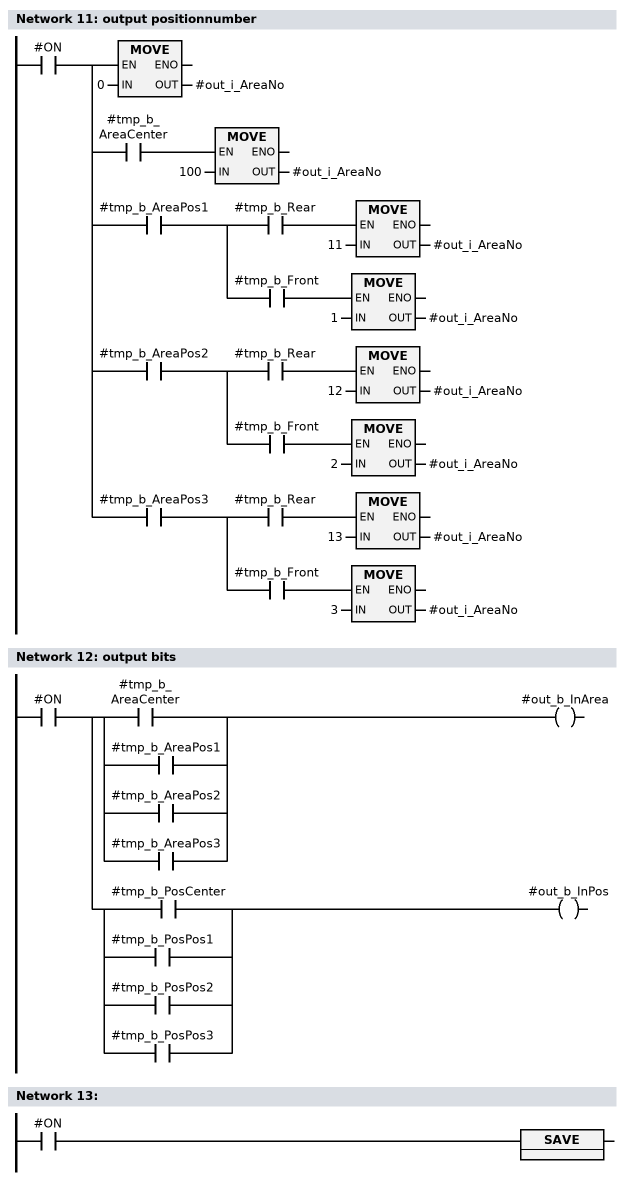
NETWORK
TITLE = output positionnumber
      A     #ON;
      =     L 10.0;
      A     L 10.0;
      JNB   _003;
      L     0;
      T     #out_i_AreaNo;
_003: NOP   0;
      A     L 10.0;
      A     #tmp_b_AreaCenter;
      JNB   _004;
      L     100;
      T     #out_i_AreaNo;
_004: NOP   0;
      A     L 10.0;
      A     #tmp_b_AreaPos1;
      =     L 10.1;
      A     L 10.1;
      A     #tmp_b_Rear;
      JNB   _005;
      L     11;
      T     #out_i_AreaNo;
_005: NOP   0;
      A     L 10.1;
      A     #tmp_b_Front;
      JNB   _006;
      L     1;
      T     #out_i_AreaNo;
_006: NOP   0;
      A     L 10.0;
      A     #tmp_b_AreaPos2;
      =     L 10.1;
      A     L 10.1;
      A     #tmp_b_Rear;
      JNB   _007;
      L     12;
      T     #out_i_AreaNo;
_007: NOP   0;
      A     L 10.1;
      A     #tmp_b_Front;
      JNB   _008;
      L     2;
      T     #out_i_AreaNo;
_008: NOP   0;
      A     L 10.0;
      A     #tmp_b_AreaPos3;
      =     L 10.1;
      A     L 10.1;
      A     #tmp_b_Rear;
      JNB   _009;
      L     13;
      T     #out_i_AreaNo;
_009: NOP   0;
      A     L 10.1;
      A     #tmp_b_Front;
      JNB   _00a;
      L     3;
      T     #out_i_AreaNo;
_00a: NOP   0;
NETWORK
TITLE = output bits
      A     #ON;
      =     L 10.0;
      A     L 10.0;
      A(;
      O     #tmp_b_AreaCenter;
      O     #tmp_b_AreaPos1;
      O     #tmp_b_AreaPos2;
      O     #tmp_b_AreaPos3;
      );
      =     #out_b_InArea;
      A     L 10.0;
      A(;
      O     #tmp_b_PosCenter;
      O     #tmp_b_PosPos1;
      O     #tmp_b_PosPos2;
      O     #tmp_b_PosPos3;
      );
      =     #out_b_InPos;
NETWORK
TITLE =
      A     #ON;
      SAVE;
END_FUNCTION

FUNCTION "Scan_TEL_Man" : VOID	// FC 28
TITLE = scan positions TELescopes manual mode
VERSION : 1.0
VAR_INPUT
  in_i_DBNo : INT ;
  in_i_NoOfDataSets : INT ;
  in_i_DatSetLenght : INT ;
  in_i_DataStartByte : INT ;
  in_di_ActAxisPos : DINT ;
  in_di_PosValMin : DINT ;
  in_di_PosValMax : DINT ;
END_VAR
VAR_OUTPUT
  out_di_PrevPos : DINT ;
  out_di_ActPos : DINT ;
  out_di_NextPos : DINT ;
  out_di_MinPos : DINT ;
  out_di_MaxPos : DINT ;
END_VAR
VAR_TEMP
  tmp_di_1 : DINT ;
  tmp_di_Pointer : DINT ;
  tmp_di_ChkPosVal : DINT ;
  tmp_di_PosData : DINT ;
  tmp_di_PosDataPlus : DINT ;
  tmp_di_PosDataMinus : DINT ;
  tmp_di_PosDataLow : DINT ;
  tmp_di_PosDataHigh : DINT ;
  tmp_di_PrevPos : DINT ;
  tmp_di_NextPos : DINT ;
  tmp_di_MinPos : DINT ;
  tmp_di_MaxPos : DINT ;
  tmp_di_TEL_in : DINT ;
  tmp_di_TEL_mid : DINT ;
  tmp_di_TEL_out : DINT ;
  tmp_i_NoOfDataSets : INT ;
  tmp_i_Counter : INT ;
  tmp_i_DBNo : INT ;
  ON : BOOL ;
  OFF : BOOL ;
END_VAR
BEGIN
NETWORK
TITLE = on/off
      SET;
      =     #ON;
      CLR;
      =     #OFF;
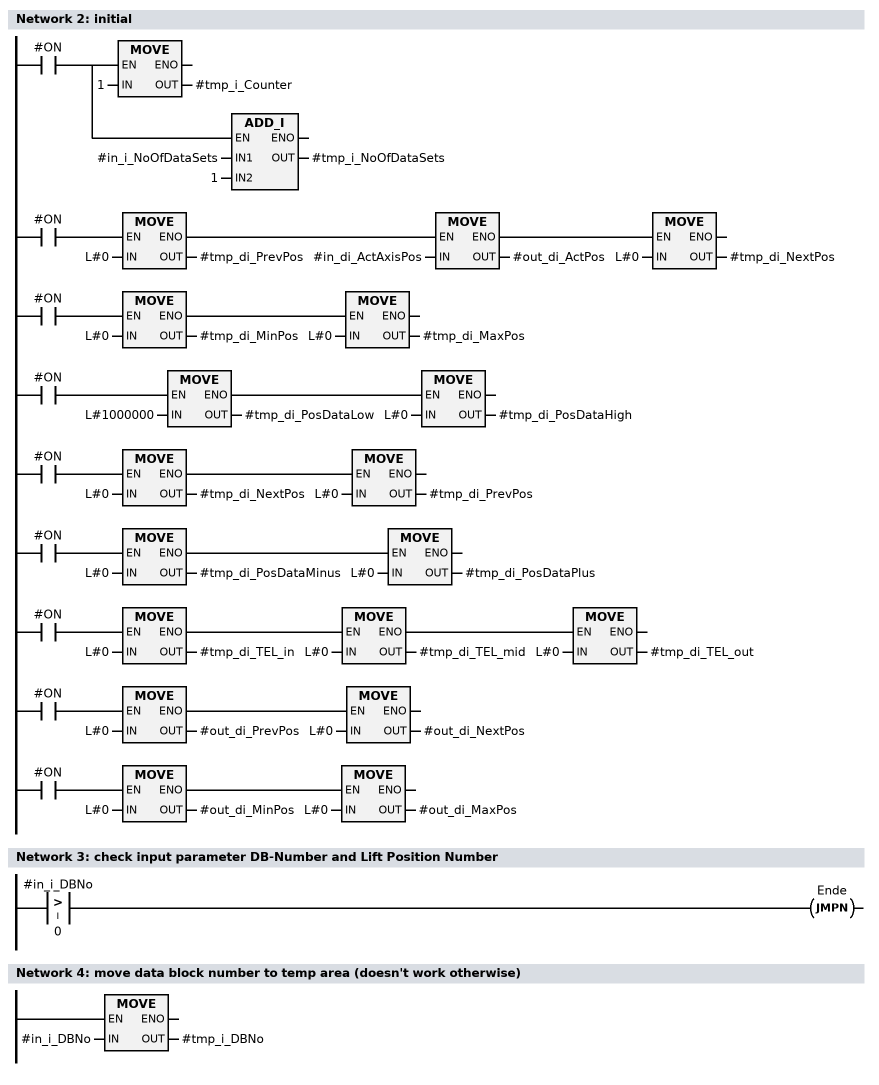
NETWORK
TITLE = initial
//set loopcounter to 0
//reset outputs
      A     #ON;
      =     L 67.0;
      A     L 67.0;
      JNB   _001;
      L     1;
      T     #tmp_i_Counter;
_001: NOP   0;
      A(;
      A(;
      A     L 67.0;
      JNB   _002;
      L     L#0;
      T     #tmp_di_PrevPos;
      SET;
      SAVE;
      CLR;
_002: A     BR;
      );
      JNB   _003;
      L     #in_di_ActAxisPos;
      T     #out_di_ActPos;
      SET;
      SAVE;
      CLR;
_003: A     BR;
      );
      JNB   _004;
      L     L#0;
      T     #tmp_di_NextPos;
_004: NOP   0;
      A(;
      A     L 67.0;
      JNB   _005;
      L     L#0;
      T     #tmp_di_MinPos;
      SET;
      SAVE;
      CLR;
_005: A     BR;
      );
      JNB   _006;
      L     L#0;
      T     #tmp_di_MaxPos;
_006: NOP   0;
      A(;
      A     L 67.0;
      JNB   _007;
      L     L#1000000;
      T     #tmp_di_PosDataLow;
      SET;
      SAVE;
      CLR;
_007: A     BR;
      );
      JNB   _008;
      L     L#0;
      T     #tmp_di_PosDataHigh;
_008: NOP   0;
      A(;
      A     L 67.0;
      JNB   _009;
      L     L#0;
      T     #tmp_di_NextPos;
      SET;
      SAVE;
      CLR;
_009: A     BR;
      );
      JNB   _00a;
      L     L#0;
      T     #tmp_di_PrevPos;
_00a: NOP   0;
      A(;
      A     L 67.0;
      JNB   _00b;
      L     L#0;
      T     #tmp_di_PosDataMinus;
      SET;
      SAVE;
      CLR;
_00b: A     BR;
      );
      JNB   _00c;
      L     L#0;
      T     #tmp_di_PosDataPlus;
_00c: NOP   0;
      A(;
      A(;
      A     L 67.0;
      JNB   _00d;
      L     L#0;
      T     #tmp_di_TEL_in;
      SET;
      SAVE;
      CLR;
_00d: A     BR;
      );
      JNB   _00e;
      L     L#0;
      T     #tmp_di_TEL_mid;
      SET;
      SAVE;
      CLR;
_00e: A     BR;
      );
      JNB   _00f;
      L     L#0;
      T     #tmp_di_TEL_out;
_00f: NOP   0;
      A     L 67.0;
      JNB   _010;
      L     #in_i_NoOfDataSets;
      L     1;
      +I;
      T     #tmp_i_NoOfDataSets;
_010: NOP   0;
      A(;
      A     L 67.0;
      JNB   _011;
      L     L#0;
      T     #out_di_PrevPos;
      SET;
      SAVE;
      CLR;
_011: A     BR;
      );
      JNB   _012;
      L     L#0;
      T     #out_di_NextPos;
_012: NOP   0;
      A(;
      A     L 67.0;
      JNB   _013;
      L     L#0;
      T     #out_di_MinPos;
      SET;
      SAVE;
      CLR;
_013: A     BR;
      );
      JNB   _014;
      L     L#0;
      T     #out_di_MaxPos;
_014: NOP   0;
NETWORK
TITLE = check input parameter DB-Number and Lift Position Number
//DB-Number > 0 and Lift in valid position
//or
//Lift position is intern hook
      L     #in_i_DBNo;
      L     0;
      >I;
      JCN   Ende;
NETWORK
TITLE = move data block number to temp area (doesn't work otherwise)
//doesn't work otherwise
      L     #in_i_DBNo;
      T     #tmp_i_DBNo;
      NOP   0;
NETWORK
TITLE = open DB
      OPN   DB [#tmp_i_DBNo];
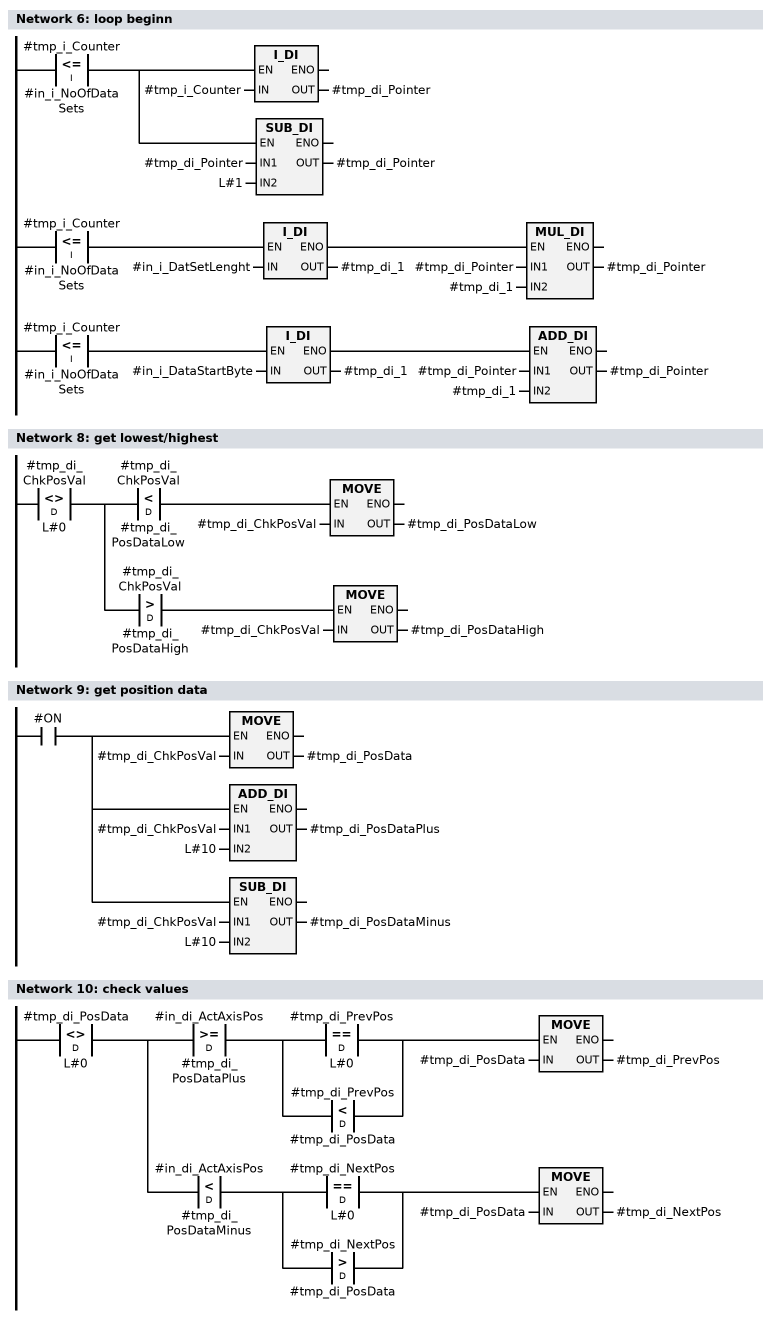
NETWORK
TITLE = loop beginn
//calculate pointer to positionvalue
scbr: L     #tmp_i_Counter;
      L     #in_i_NoOfDataSets;
      <=I;
      =     L 67.0;
      A     L 67.0;
      JNB   _015;
      L     #tmp_i_Counter;
      ITD;
      T     #tmp_di_Pointer;
_015: NOP   0;
      A     L 67.0;
      JNB   _016;
      L     #tmp_di_Pointer;
      L     L#1;
      -D;
      T     #tmp_di_Pointer;
_016: NOP   0;
      A(;
      A     L 67.0;
      JNB   _017;
      L     #in_i_DatSetLenght;
      ITD;
      T     #tmp_di_1;
      SET;
      SAVE;
      CLR;
_017: A     BR;
      );
      JNB   _018;
      L     #tmp_di_Pointer;
      L     #tmp_di_1;
      *D;
      T     #tmp_di_Pointer;
_018: NOP   0;
      A(;
      A     L 67.0;
      JNB   _019;
      L     #in_i_DataStartByte;
      ITD;
      T     #tmp_di_1;
      SET;
      SAVE;
      CLR;
_019: A     BR;
      );
      JNB   _01a;
      L     #tmp_di_Pointer;
      L     #tmp_di_1;
      +D;
      T     #tmp_di_Pointer;
_01a: NOP   0;
NETWORK
TITLE = get positionvalue
      L     #tmp_di_Pointer;	// load pointer
      SLD   3;	// shift left 3 bits to achieve pointer format
      LAR1;	// load adressregister 1 with pointer
      L     DBD [AR1,P#0.0];	// load position from DataBlock
      T     #tmp_di_ChkPosVal;
NETWORK
TITLE = get lowest/highest
      L     #tmp_di_ChkPosVal;
      L     L#0;
      <>D;
      =     L 67.0;
      A     L 67.0;
      A(;
      L     #tmp_di_ChkPosVal;
      L     #tmp_di_PosDataLow;
      <D;
      );
      JNB   _01b;
      L     #tmp_di_ChkPosVal;
      T     #tmp_di_PosDataLow;
_01b: NOP   0;
      A     L 67.0;
      A(;
      L     #tmp_di_ChkPosVal;
      L     #tmp_di_PosDataHigh;
      >D;
      );
      JNB   _01c;
      L     #tmp_di_ChkPosVal;
      T     #tmp_di_PosDataHigh;
_01c: NOP   0;
NETWORK
TITLE = get position data
      A     #ON;
      =     L 67.0;
      A     L 67.0;
      JNB   _01d;
      L     #tmp_di_ChkPosVal;
      T     #tmp_di_PosData;
_01d: NOP   0;
      A     L 67.0;
      JNB   _01e;
      L     #tmp_di_ChkPosVal;
      L     L#10;
      +D;
      T     #tmp_di_PosDataPlus;
_01e: NOP   0;
      A     L 67.0;
      JNB   _01f;
      L     #tmp_di_ChkPosVal;
      L     L#10;
      -D;
      T     #tmp_di_PosDataMinus;
_01f: NOP   0;
NETWORK
TITLE = check values
      L     #tmp_di_PosData;
      L     L#0;
      <>D;
      =     L 67.0;
      A     L 67.0;
      A(;
      L     #in_di_ActAxisPos;
      L     #tmp_di_PosDataPlus;
      >=D;
      );
      A(;
      O(;
      L     #tmp_di_PrevPos;
      L     L#0;
      ==D;
      );
      O(;
      L     #tmp_di_PrevPos;
      L     #tmp_di_PosData;
      <D;
      );
      );
      JNB   _020;
      L     #tmp_di_PosData;
      T     #tmp_di_PrevPos;
_020: NOP   0;
      A     L 67.0;
      A(;
      L     #in_di_ActAxisPos;
      L     #tmp_di_PosDataMinus;
      <D;
      );
      A(;
      O(;
      L     #tmp_di_NextPos;
      L     L#0;
      ==D;
      );
      O(;
      L     #tmp_di_NextPos;
      L     #tmp_di_PosData;
      >D;
      );
      );
      JNB   _021;
      L     #tmp_di_PosData;
      T     #tmp_di_NextPos;
_021: NOP   0;
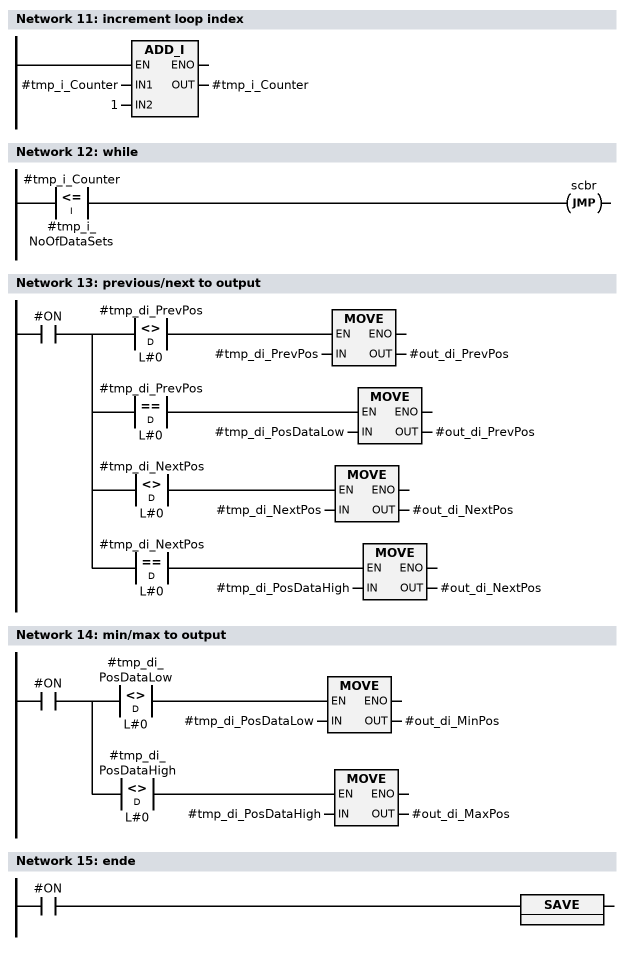
NETWORK
TITLE = increment loop index
      L     #tmp_i_Counter;
      L     1;
      +I;
      T     #tmp_i_Counter;
      NOP   0;
NETWORK
TITLE = while 
      L     #tmp_i_Counter;
      L     #tmp_i_NoOfDataSets;
      <=I;
      JC    scbr;
NETWORK
TITLE = previous/next to output
Ende: A     #ON;
      =     L 67.0;
      A     L 67.0;
      A(;
      L     #tmp_di_PrevPos;
      L     L#0;
      <>D;
      );
      JNB   _022;
      L     #tmp_di_PrevPos;
      T     #out_di_PrevPos;
_022: NOP   0;
      A     L 67.0;
      A(;
      L     #tmp_di_PrevPos;
      L     L#0;
      ==D;
      );
      JNB   _023;
      L     #tmp_di_PosDataLow;
      T     #out_di_PrevPos;
_023: NOP   0;
      A     L 67.0;
      A(;
      L     #tmp_di_NextPos;
      L     L#0;
      <>D;
      );
      JNB   _024;
      L     #tmp_di_NextPos;
      T     #out_di_NextPos;
_024: NOP   0;
      A     L 67.0;
      A(;
      L     #tmp_di_NextPos;
      L     L#0;
      ==D;
      );
      JNB   _025;
      L     #tmp_di_PosDataHigh;
      T     #out_di_NextPos;
_025: NOP   0;
NETWORK
TITLE = min/max to output
      A     #ON;
      =     L 67.0;
      A     L 67.0;
      A(;
      L     #tmp_di_PosDataLow;
      L     L#0;
      <>D;
      );
      JNB   _026;
      L     #tmp_di_PosDataLow;
      T     #out_di_MinPos;
_026: NOP   0;
      A     L 67.0;
      A(;
      L     #tmp_di_PosDataHigh;
      L     L#0;
      <>D;
      );
      JNB   _027;
      L     #tmp_di_PosDataHigh;
      T     #out_di_MaxPos;
_027: NOP   0;
NETWORK
TITLE = ende
      A     #ON;
      SAVE;
END_FUNCTION

FUNCTION "SCALE_WAGO_AI" : WORD	// FC 29
TITLE = SCALING VALUES
//Speziell für WAGO 250-466 4.20mA SE standard 
//Meßwertauflösung 12 bit (4095)
//
AUTHOR : SEA
FAMILY : CONVERT
NAME : SCALE
VERSION : 2.1
VAR_INPUT
  IN : INT ;	// input value to be scaled
  HI_LIM : REAL ;	// upper limit in engineering units
  LO_LIM : REAL ;	// lower limit in engineering units
  BIPOLAR : BOOL ;	// 1=bipolar; 0=unipolar
END_VAR
VAR_OUTPUT
  RET_VAL : WORD ;
  OUT : REAL ;	// result of the scale conversion
END_VAR
VAR_TEMP
  IN_REAL : REAL ;	// input value as a REAL number
  K1 : REAL ;	// low limit for input value
  K2 : REAL ;	// high limit for input value
  SPAN : REAL ;	// HI_LIM - LO_LIM
  TEMP1 : REAL ;	// temporary result
END_VAR
BEGIN
NETWORK
TITLE =
//
// set K1 and K2 constants based upon BIPOLAR
//
// (network holds code this reader does not know; not shown)
// convert input (IN) to real
// determine SPAN = HI_LIM - LO_LIM
// If the input value is outside the K1 and K2 range, the output
// is clamped to the nearer of either the LO_LIM or the HI_LIM 
// and an error is logged. If the input value is exactly at a limit the
// output will be set to the computed limit with no error returned.
//     changed 2/14/00 by ERI per RQ210693
// scale the input
// set BR bit : no error-set BR bit to 1; with error-set BR bit to 0.
END_FUNCTION

FUNCTION "Inputs" : VOID	// FC 30
TITLE = Inputs
VERSION : 0.1
VAR_TEMP
  tmp_Retval : INT ;
  tmp_d : INT ;
  tmp_u : DINT ;
  value : INT ;
  d_value : DINT ;
  ON : BOOL ;
  OFF : BOOL ;
  tmp_in : DINT ;
END_VAR
BEGIN
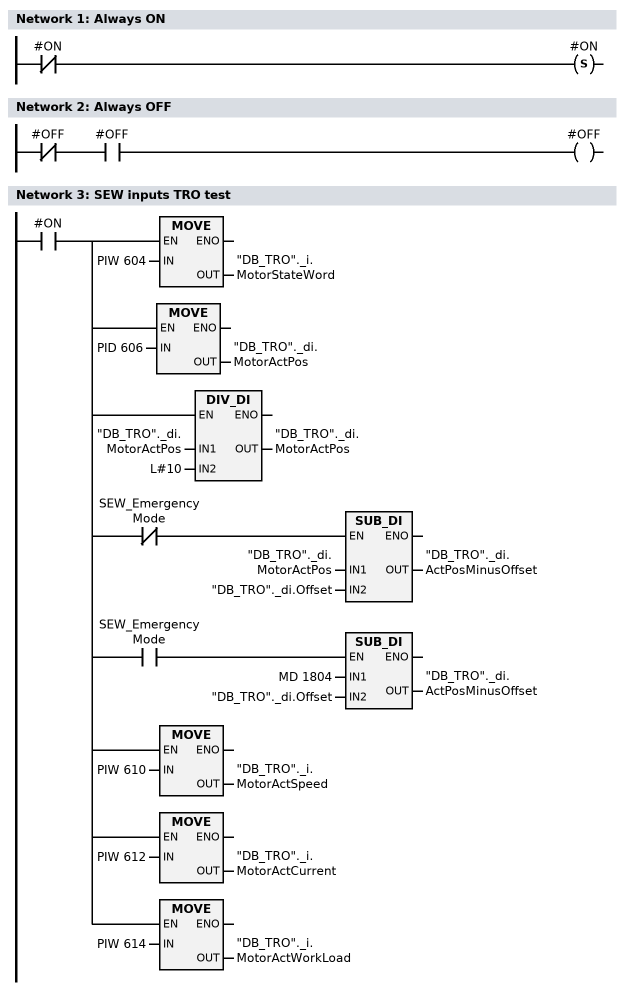
NETWORK
TITLE = Always ON
      AN    #ON;
      S     #ON;
NETWORK
TITLE = Always OFF
      AN    #OFF;
      A     #OFF;
      =     #OFF;
NETWORK
TITLE = SEW inputs TRO test
      A     #ON;
      =     L 20.0;
      A     L 20.0;
      JNB   _001;
      L     PIW 604;
      T     "DB_TRO"._i.MotorStateWord;
_001: NOP   0;
      A     L 20.0;
      JNB   _002;
      L     PID 606;
      T     "DB_TRO"._di.MotorActPos;
_002: NOP   0;
      A     L 20.0;
      JNB   _003;
      L     "DB_TRO"._di.MotorActPos;
      L     L#10;
      /D;
      T     "DB_TRO"._di.MotorActPos;
_003: NOP   0;
      A     L 20.0;
      AN    "SEW_EmergencyMode";
      JNB   _004;
      L     "DB_TRO"._di.MotorActPos;
      L     "DB_TRO"._di.Offset;
      -D;
      T     "DB_TRO"._di.ActPosMinusOffset;
_004: NOP   0;
      A     L 20.0;
      A     "SEW_EmergencyMode";
      JNB   _005;
      L     MD 1804;
      L     "DB_TRO"._di.Offset;
      -D;
      T     "DB_TRO"._di.ActPosMinusOffset;
_005: NOP   0;
      A     L 20.0;
      JNB   _006;
      L     PIW 610;
      T     "DB_TRO"._i.MotorActSpeed;
_006: NOP   0;
      A     L 20.0;
      JNB   _007;
      L     PIW 612;
      T     "DB_TRO"._i.MotorActCurrent;
_007: NOP   0;
      A     L 20.0;
      JNB   _008;
      L     PIW 614;
      T     "DB_TRO"._i.MotorActWorkLoad;
_008: NOP   0;
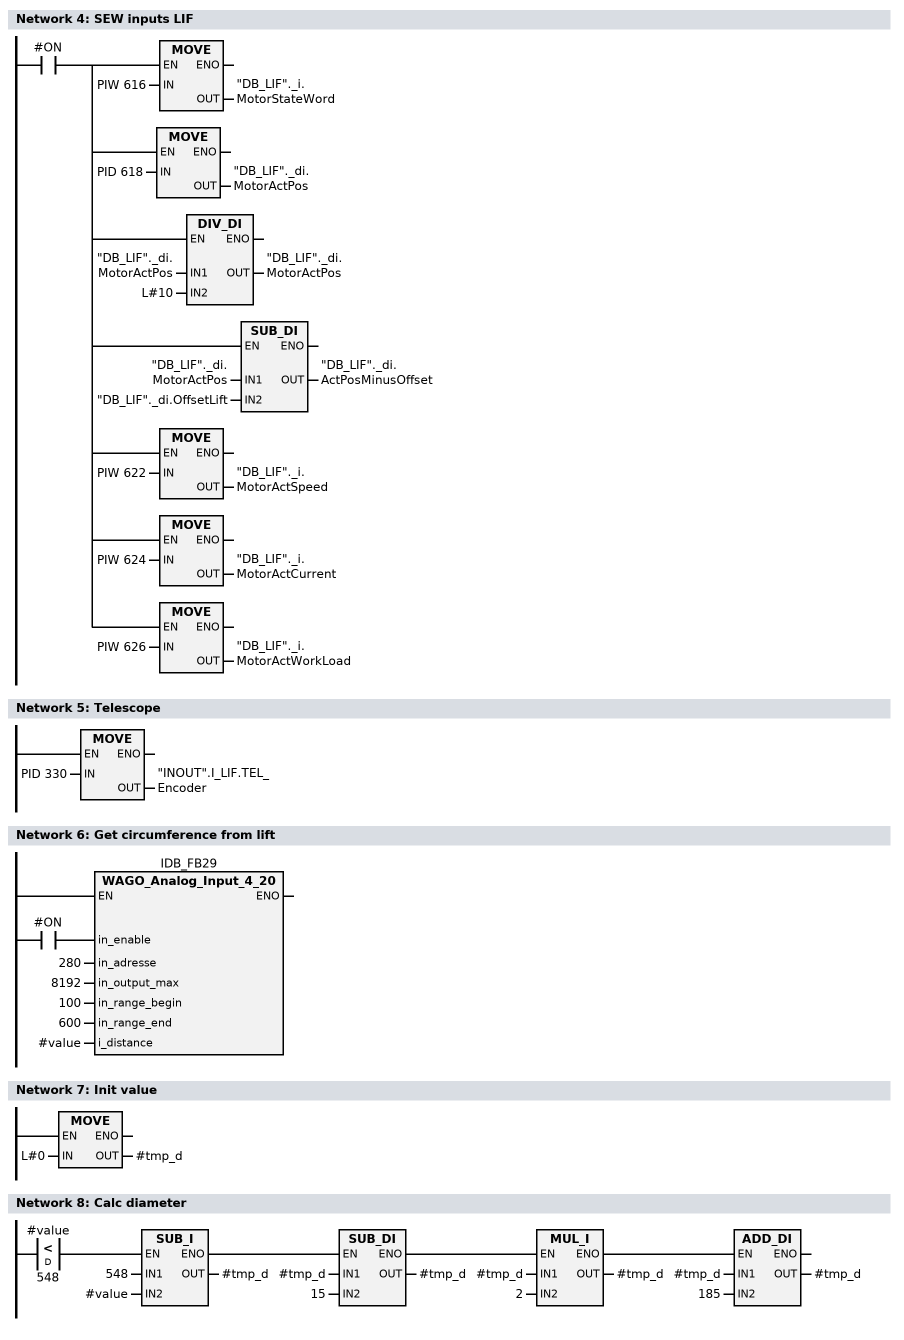
NETWORK
TITLE = SEW inputs LIF
      A     #ON;
      =     L 20.0;
      A     L 20.0;
      JNB   _009;
      L     PIW 616;
      T     "DB_LIF"._i.MotorStateWord;
_009: NOP   0;
      A     L 20.0;
      JNB   _00a;
      L     PID 618;
      T     "DB_LIF"._di.MotorActPos;
_00a: NOP   0;
      A     L 20.0;
      JNB   _00b;
      L     "DB_LIF"._di.MotorActPos;
      L     L#10;
      /D;
      T     "DB_LIF"._di.MotorActPos;
_00b: NOP   0;
      A     L 20.0;
      JNB   _00c;
      L     "DB_LIF"._di.MotorActPos;
      L     "DB_LIF"._di.OffsetLift;
      -D;
      T     "DB_LIF"._di.ActPosMinusOffset;
_00c: NOP   0;
      A     L 20.0;
      JNB   _00d;
      L     PIW 622;
      T     "DB_LIF"._i.MotorActSpeed;
_00d: NOP   0;
      A     L 20.0;
      JNB   _00e;
      L     PIW 624;
      T     "DB_LIF"._i.MotorActCurrent;
_00e: NOP   0;
      A     L 20.0;
      JNB   _00f;
      L     PIW 626;
      T     "DB_LIF"._i.MotorActWorkLoad;
_00f: NOP   0;
NETWORK
TITLE = Telescope
//we use a offset 10000
//
//bc17.02.2019: nachrüstung Encoder
//
      L     PID 330;
      T     "INOUT".I_LIF.TEL_Encoder;
      NOP   0;
NETWORK
TITLE = Get circumference from lift
//100mm = A1 Setpoint
//600mm = A2 Setpoint
//with pipe = 548
//US setting BEAM = 2
      A     #ON;
      =     L 20.0;
      BLD   103;
      CALL  "WAGO_Analog_Input_4_20" , "IDB_FB29" (
           in_enable                := L 20.0,
           in_adresse               := 280,
           in_output_max            := 8192,
           in_range_begin           := 100,
           in_range_end             := 600,
           i_distance               := #value);
      NOP   0;
NETWORK
TITLE = Init value
      L     L#0;
      T     #tmp_d;
      NOP   0;
NETWORK
TITLE = Calc diameter
//calc (548 - value - core thickness) * 2 + core diameter
      A(;
      A(;
      A(;
      A(;
      L     #value;
      L     548;
      <D;
      );
      JNB   _010;
      L     548;
      L     #value;
      -I;
      T     #tmp_d;
      AN    OV;
      SAVE;
      CLR;
_010: A     BR;
      );
      JNB   _011;
      L     #tmp_d;
      L     15;
      -D;
      T     #tmp_d;
      AN    OV;
      SAVE;
      CLR;
_011: A     BR;
      );
      JNB   _012;
      L     #tmp_d;
      L     2;
      *I;
      T     #tmp_d;
      AN    OV;
      SAVE;
      CLR;
_012: A     BR;
      );
      JNB   _013;
      L     #tmp_d;
      L     185;
      +D;
      T     #tmp_d;
_013: NOP   0;
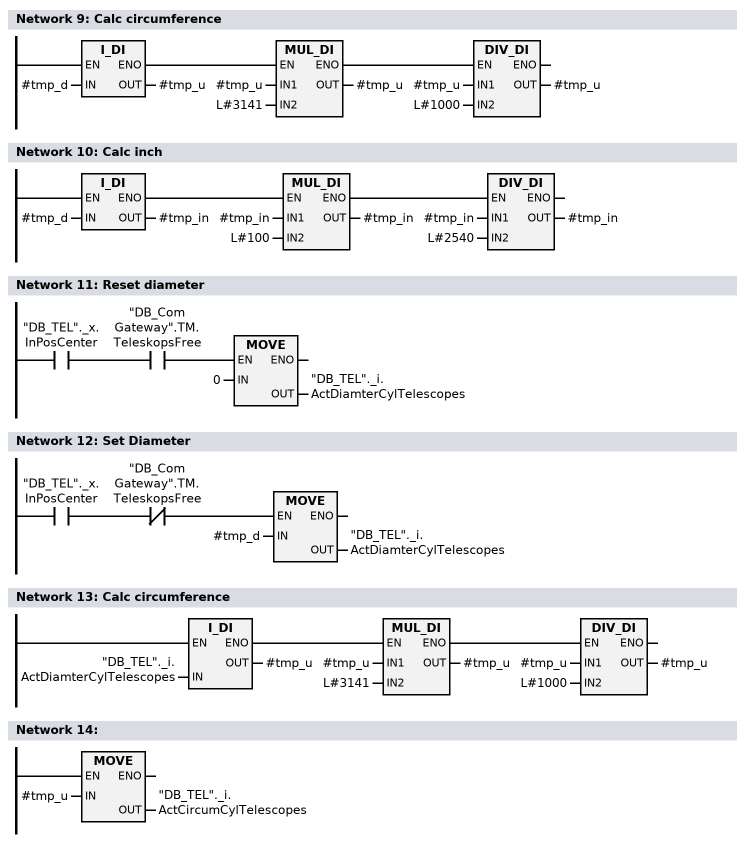
NETWORK
TITLE = Calc circumference
      A(;
      A(;
      L     #tmp_d;
      ITD;
      T     #tmp_u;
      SET;
      SAVE;
      CLR;
      A     BR;
      );
      JNB   _014;
      L     #tmp_u;
      L     L#3141;
      *D;
      T     #tmp_u;
      AN    OV;
      SAVE;
      CLR;
_014: A     BR;
      );
      JNB   _015;
      L     #tmp_u;
      L     L#1000;
      /D;
      T     #tmp_u;
_015: NOP   0;
NETWORK
TITLE = Calc inch
//25.4 mm = 1 inch 
//
//40 inch = 1016
//34 inch = 863
//14 inch = 355 330
      A(;
      A(;
      L     #tmp_d;
      ITD;
      T     #tmp_in;
      SET;
      SAVE;
      CLR;
      A     BR;
      );
      JNB   _016;
      L     #tmp_in;
      L     L#100;
      *D;
      T     #tmp_in;
      AN    OV;
      SAVE;
      CLR;
_016: A     BR;
      );
      JNB   _017;
      L     #tmp_in;
      L     L#2540;
      /D;
      T     #tmp_in;
_017: NOP   0;
NETWORK
TITLE = Reset diameter
      A     "DB_TEL"._x.InPosCenter;
      A     "DB_ComGateway".TM.TeleskopsFree;
      JNB   _018;
      L     0;
      T     "DB_TEL"._i.ActDiamterCylTelescopes;
_018: NOP   0;
NETWORK
TITLE = Set Diameter
      A     "DB_TEL"._x.InPosCenter;
      AN    "DB_ComGateway".TM.TeleskopsFree;
      JNB   _019;
      L     #tmp_d;
      T     "DB_TEL"._i.ActDiamterCylTelescopes;
_019: NOP   0;
NETWORK
TITLE = Calc circumference
      A(;
      A(;
      L     "DB_TEL"._i.ActDiamterCylTelescopes;
      ITD;
      T     #tmp_u;
      SET;
      SAVE;
      CLR;
      A     BR;
      );
      JNB   _01a;
      L     #tmp_u;
      L     L#3141;
      *D;
      T     #tmp_u;
      AN    OV;
      SAVE;
      CLR;
_01a: A     BR;
      );
      JNB   _01b;
      L     #tmp_u;
      L     L#1000;
      /D;
      T     #tmp_u;
_01b: NOP   0;
NETWORK
TITLE =
      L     #tmp_u;
      T     "DB_TEL"._i.ActCircumCylTelescopes;
      NOP   0;
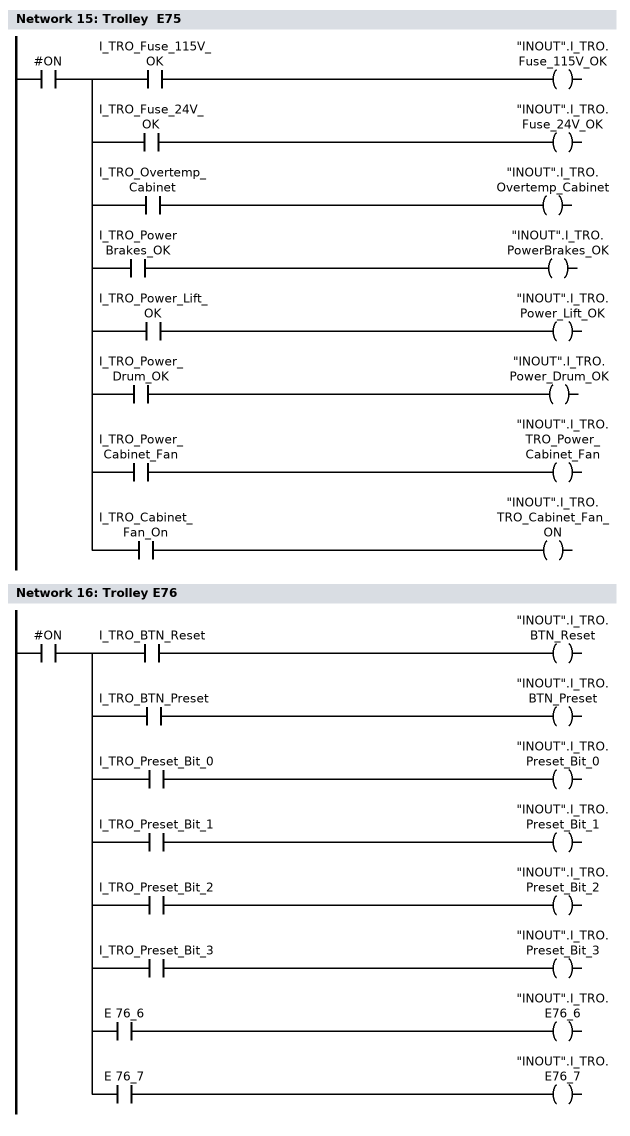
NETWORK
TITLE = Trolley  E75
      A     #ON;
      =     L 20.0;
      A     L 20.0;
      A     "I_TRO_Fuse_115V_OK";
      =     "INOUT".I_TRO.Fuse_115V_OK;
      A     L 20.0;
      A     "I_TRO_Fuse_24V_OK";
      =     "INOUT".I_TRO.Fuse_24V_OK;
      A     L 20.0;
      A     "I_TRO_Overtemp_Cabinet";
      =     "INOUT".I_TRO.Overtemp_Cabinet;
      A     L 20.0;
      A     "I_TRO_Power Brakes_OK";
      =     "INOUT".I_TRO.PowerBrakes_OK;
      A     L 20.0;
      A     "I_TRO_Power_Lift_OK";
      =     "INOUT".I_TRO.Power_Lift_OK;
      A     L 20.0;
      A     "I_TRO_Power_Drum_OK";
      =     "INOUT".I_TRO.Power_Drum_OK;
      A     L 20.0;
      A     "I_TRO_Power_Cabinet_Fan";
      =     "INOUT".I_TRO.TRO_Power_Cabinet_Fan;
      A     L 20.0;
      A     "I_TRO_Cabinet_Fan_On";
      =     "INOUT".I_TRO.TRO_Cabinet_Fan_ON;
NETWORK
TITLE = Trolley E76 
      A     #ON;
      =     L 20.0;
      A     L 20.0;
      A     "I_TRO_BTN_Reset";
      =     "INOUT".I_TRO.BTN_Reset;
      A     L 20.0;
      A     "I_TRO_BTN_Preset";
      =     "INOUT".I_TRO.BTN_Preset;
      A     L 20.0;
      A     "I_TRO_Preset_Bit_0";
      =     "INOUT".I_TRO.Preset_Bit_0;
      A     L 20.0;
      A     "I_TRO_Preset_Bit_1";
      =     "INOUT".I_TRO.Preset_Bit_1;
      A     L 20.0;
      A     "I_TRO_Preset_Bit_2";
      =     "INOUT".I_TRO.Preset_Bit_2;
      A     L 20.0;
      A     "I_TRO_Preset_Bit_3";
      =     "INOUT".I_TRO.Preset_Bit_3;
      A     L 20.0;
      A     "E 76_6";
      =     "INOUT".I_TRO.E76_6;
      A     L 20.0;
      A     "E 76_7";
      =     "INOUT".I_TRO.E76_7;
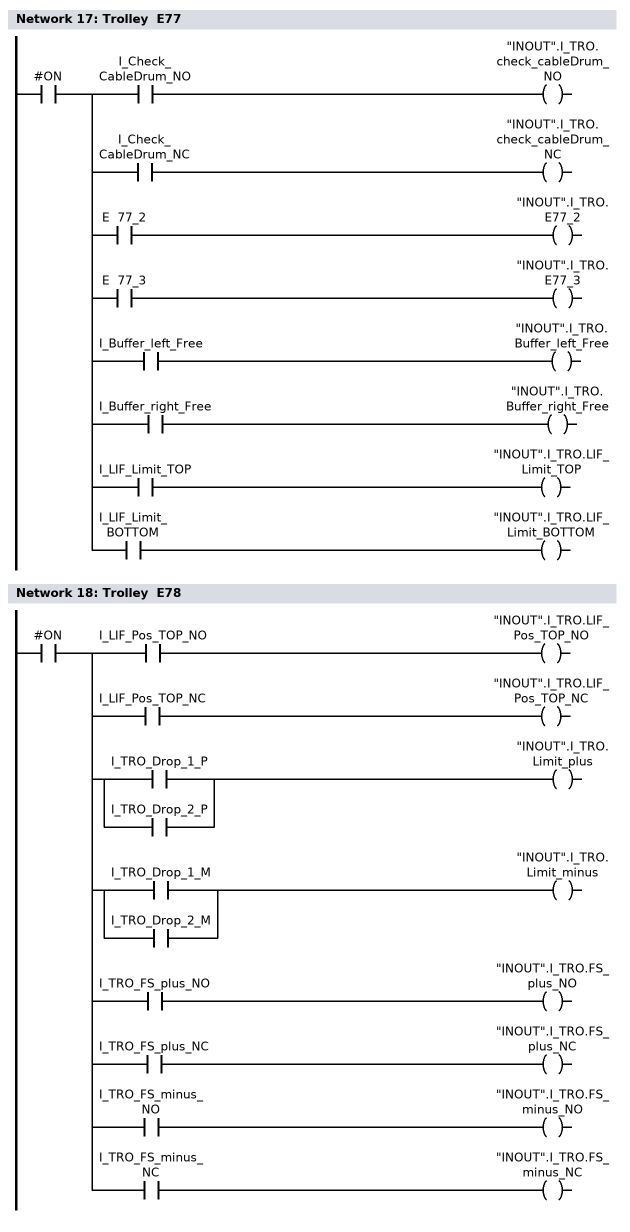
NETWORK
TITLE = Trolley  E77
      A     #ON;
      =     L 20.0;
      A     L 20.0;
      A     "I_Check_CableDrum_NO";
      =     "INOUT".I_TRO.check_cableDrum_NO;
      A     L 20.0;
      A     "I_Check_CableDrum_NC";
      =     "INOUT".I_TRO.check_cableDrum_NC;
      A     L 20.0;
      A     "E  77_2";
      =     "INOUT".I_TRO.E77_2;
      A     L 20.0;
      A     "E  77_3";
      =     "INOUT".I_TRO.E77_3;
      A     L 20.0;
      A     "I_Buffer_left_Free";
      =     "INOUT".I_TRO.Buffer_left_Free;
      A     L 20.0;
      A     "I_Buffer_right_Free";
      =     "INOUT".I_TRO.Buffer_right_Free;
      A     L 20.0;
      A     "I_LIF_Limit_TOP";
      =     "INOUT".I_TRO.LIF_Limit_TOP;
      A     L 20.0;
      A     "I_LIF_Limit_BOTTOM";
      =     "INOUT".I_TRO.LIF_Limit_BOTTOM;
NETWORK
TITLE = Trolley  E78
      A     #ON;
      =     L 20.0;
      A     L 20.0;
      A     "I_LIF_Pos_TOP_NO";
      =     "INOUT".I_TRO.LIF_Pos_TOP_NO;
      A     L 20.0;
      A     "I_LIF_Pos_TOP_NC";
      =     "INOUT".I_TRO.LIF_Pos_TOP_NC;
      A     L 20.0;
      A(;
      O     "I_TRO_Drop_1_P";
      O     "I_TRO_Drop_2_P";
      );
      =     "INOUT".I_TRO.Limit_plus;
      A     L 20.0;
      A(;
      O     "I_TRO_Drop_1_M";
      O     "I_TRO_Drop_2_M";
      );
      =     "INOUT".I_TRO.Limit_minus;
      A     L 20.0;
      A     "I_TRO_FS_plus_NO";
      =     "INOUT".I_TRO.FS_plus_NO;
      A     L 20.0;
      A     "I_TRO_FS_plus_NC";
      =     "INOUT".I_TRO.FS_plus_NC;
      A     L 20.0;
      A     "I_TRO_FS_minus_NO";
      =     "INOUT".I_TRO.FS_minus_NO;
      A     L 20.0;
      A     "I_TRO_FS_minus_NC";
      =     "INOUT".I_TRO.FS_minus_NC;
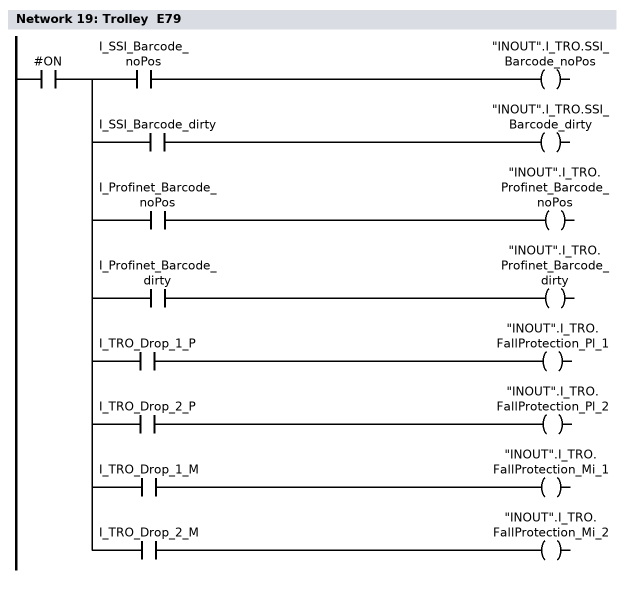
NETWORK
TITLE = Trolley  E79
      A     #ON;
      =     L 20.0;
      A     L 20.0;
      A     "I_SSI_Barcode_noPos";
      =     "INOUT".I_TRO.SSI_Barcode_noPos;
      A     L 20.0;
      A     "I_SSI_Barcode_dirty";
      =     "INOUT".I_TRO.SSI_Barcode_dirty;
      A     L 20.0;
      A     "I_Profinet_Barcode_noPos";
      =     "INOUT".I_TRO.Profinet_Barcode_noPos;
      A     L 20.0;
      A     "I_Profinet_Barcode_dirty";
      =     "INOUT".I_TRO.Profinet_Barcode_dirty;
      A     L 20.0;
      A     "I_TRO_Drop_1_P";
      =     "INOUT".I_TRO.FallProtection_Pl_1;
      A     L 20.0;
      A     "I_TRO_Drop_2_P";
      =     "INOUT".I_TRO.FallProtection_Pl_2;
      A     L 20.0;
      A     "I_TRO_Drop_1_M";
      =     "INOUT".I_TRO.FallProtection_Mi_1;
      A     L 20.0;
      A     "I_TRO_Drop_2_M";
      =     "INOUT".I_TRO.FallProtection_Mi_2;
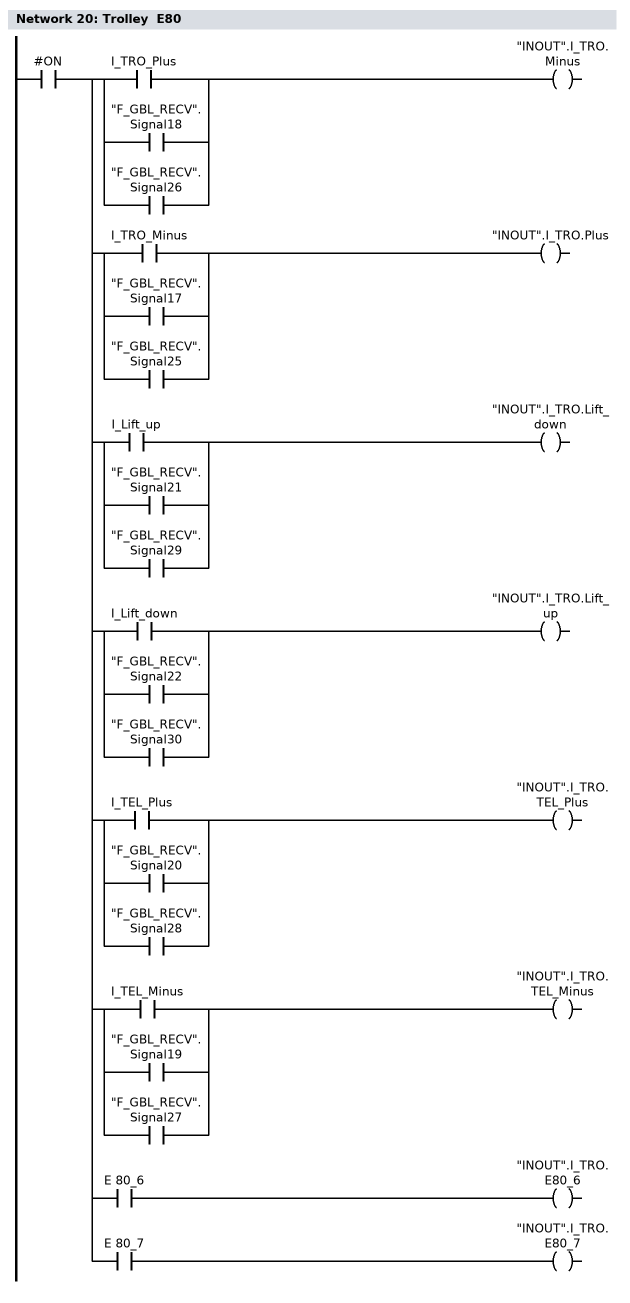
NETWORK
TITLE = Trolley  E80
      A     #ON;
      =     L 20.0;
      A     L 20.0;
      A(;
      O     "I_TRO_Plus";
      O     "F_GBL_RECV".Signal18;
      O     "F_GBL_RECV".Signal26;
      );
      =     "INOUT".I_TRO.Minus;
      A     L 20.0;
      A(;
      O     "I_TRO_Minus";
      O     "F_GBL_RECV".Signal17;
      O     "F_GBL_RECV".Signal25;
      );
      =     "INOUT".I_TRO.Plus;
      A     L 20.0;
      A(;
      O     "I_Lift_up";
      O     "F_GBL_RECV".Signal21;
      O     "F_GBL_RECV".Signal29;
      );
      =     "INOUT".I_TRO.Lift_down;
      A     L 20.0;
      A(;
      O     "I_Lift_down";
      O     "F_GBL_RECV".Signal22;
      O     "F_GBL_RECV".Signal30;
      );
      =     "INOUT".I_TRO.Lift_up;
      A     L 20.0;
      A(;
      O     "I_TEL_Plus";
      O     "F_GBL_RECV".Signal20;
      O     "F_GBL_RECV".Signal28;
      );
      =     "INOUT".I_TRO.TEL_Plus;
      A     L 20.0;
      A(;
      O     "I_TEL_Minus";
      O     "F_GBL_RECV".Signal19;
      O     "F_GBL_RECV".Signal27;
      );
      =     "INOUT".I_TRO.TEL_Minus;
      A     L 20.0;
      A     "E 80_6";
      =     "INOUT".I_TRO.E80_6;
      A     L 20.0;
      A     "E 80_7";
      =     "INOUT".I_TRO.E80_7;
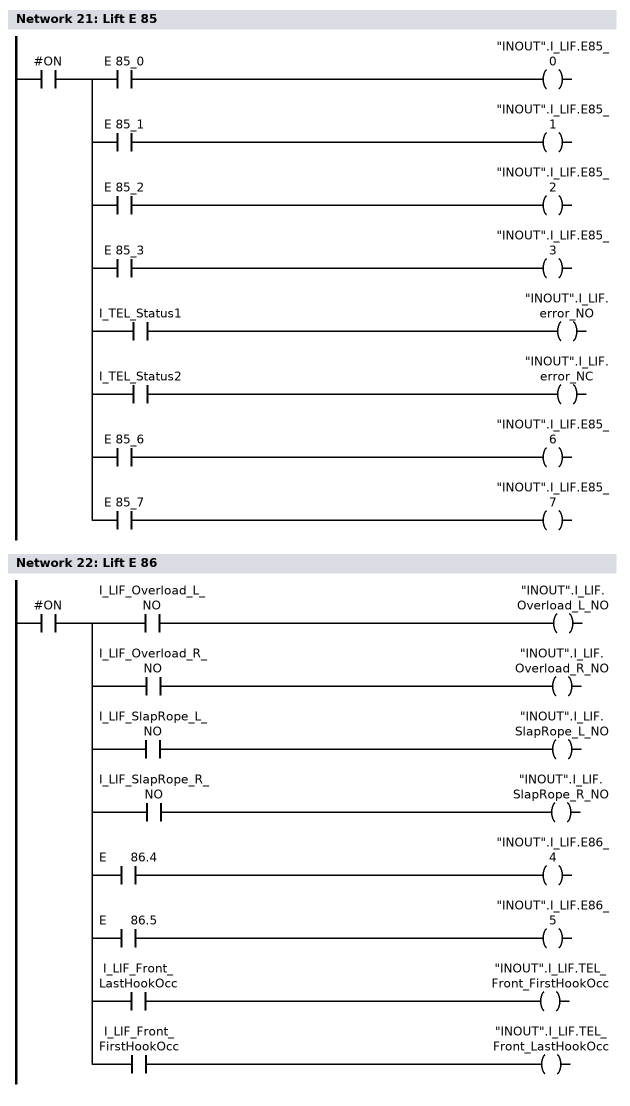
NETWORK
TITLE = Lift E 85
      A     #ON;
      =     L 20.0;
      A     L 20.0;
      A     "E 85_0";
      =     "INOUT".I_LIF.E85_0;
      A     L 20.0;
      A     "E 85_1";
      =     "INOUT".I_LIF.E85_1;
      A     L 20.0;
      A     "E 85_2";
      =     "INOUT".I_LIF.E85_2;
      A     L 20.0;
      A     "E 85_3";
      =     "INOUT".I_LIF.E85_3;
      A     L 20.0;
      A     "I_TEL_Status1";
      =     "INOUT".I_LIF.error_NO;
      A     L 20.0;
      A     "I_TEL_Status2";
      =     "INOUT".I_LIF.error_NC;
      A     L 20.0;
      A     "E 85_6";
      =     "INOUT".I_LIF.E85_6;
      A     L 20.0;
      A     "E 85_7";
      =     "INOUT".I_LIF.E85_7;
NETWORK
TITLE = Lift E 86
      A     #ON;
      =     L 20.0;
      A     L 20.0;
      A     "I_LIF_Overload_L_NO";
      =     "INOUT".I_LIF.Overload_L_NO;
      A     L 20.0;
      A     "I_LIF_Overload_R_NO";
      =     "INOUT".I_LIF.Overload_R_NO;
      A     L 20.0;
      A     "I_LIF_SlapRope_L_NO";
      =     "INOUT".I_LIF.SlapRope_L_NO;
      A     L 20.0;
      A     "I_LIF_SlapRope_R_NO";
      =     "INOUT".I_LIF.SlapRope_R_NO;
      A     L 20.0;
      A     "E      86.4";
      =     "INOUT".I_LIF.E86_4;
      A     L 20.0;
      A     "E      86.5";
      =     "INOUT".I_LIF.E86_5;
      A     L 20.0;
      A     "I_LIF_Front_LastHookOcc";
      =     "INOUT".I_LIF.TEL_Front_FirstHookOcc;
      A     L 20.0;
      A     "I_LIF_Front_FirstHookOcc";
      =     "INOUT".I_LIF.TEL_Front_LastHookOcc;
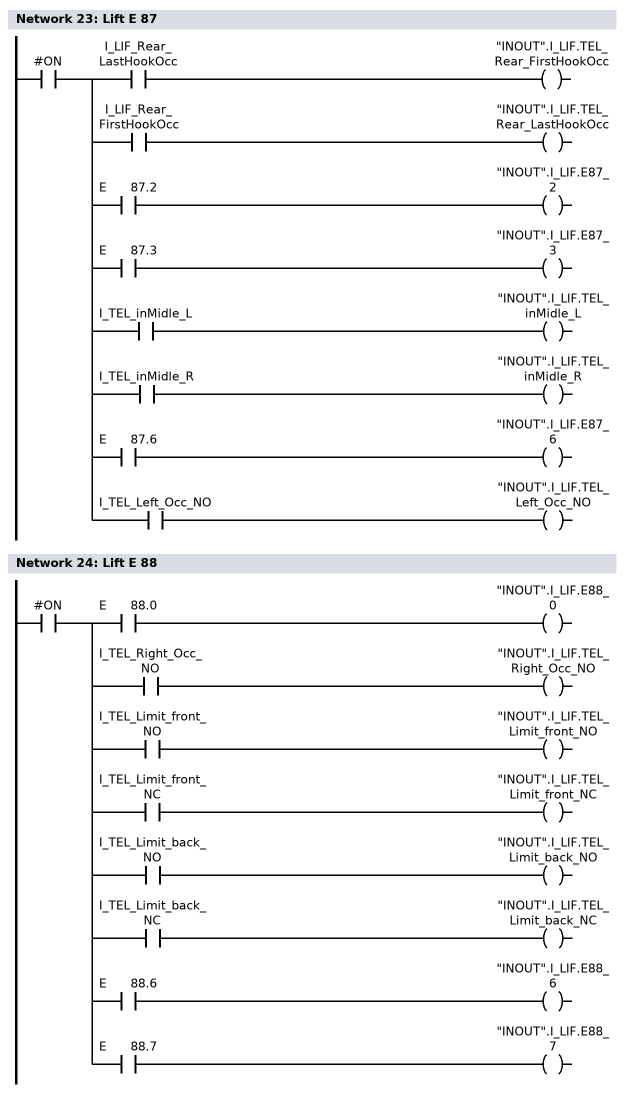
NETWORK
TITLE = Lift E 87
      A     #ON;
      =     L 20.0;
      A     L 20.0;
      A     "I_LIF_Rear_LastHookOcc";
      =     "INOUT".I_LIF.TEL_Rear_FirstHookOcc;
      A     L 20.0;
      A     "I_LIF_Rear_FirstHookOcc";
      =     "INOUT".I_LIF.TEL_Rear_LastHookOcc;
      A     L 20.0;
      A     "E      87.2";
      =     "INOUT".I_LIF.E87_2;
      A     L 20.0;
      A     "E      87.3";
      =     "INOUT".I_LIF.E87_3;
      A     L 20.0;
      A     "I_TEL_inMidle_L";
      =     "INOUT".I_LIF.TEL_inMidle_L;
      A     L 20.0;
      A     "I_TEL_inMidle_R";
      =     "INOUT".I_LIF.TEL_inMidle_R;
      A     L 20.0;
      A     "E      87.6";
      =     "INOUT".I_LIF.E87_6;
      A     L 20.0;
      A     "I_TEL_Left_Occ_NO";
      =     "INOUT".I_LIF.TEL_Left_Occ_NO;
NETWORK
TITLE = Lift E 88
      A     #ON;
      =     L 20.0;
      A     L 20.0;
      A     "E      88.0";
      =     "INOUT".I_LIF.E88_0;
      A     L 20.0;
      A     "I_TEL_Right_Occ_NO";
      =     "INOUT".I_LIF.TEL_Right_Occ_NO;
      A     L 20.0;
      A     "I_TEL_Limit_front_NO";
      =     "INOUT".I_LIF.TEL_Limit_front_NO;
      A     L 20.0;
      A     "I_TEL_Limit_front_NC";
      =     "INOUT".I_LIF.TEL_Limit_front_NC;
      A     L 20.0;
      A     "I_TEL_Limit_back_NO";
      =     "INOUT".I_LIF.TEL_Limit_back_NO;
      A     L 20.0;
      A     "I_TEL_Limit_back_NC";
      =     "INOUT".I_LIF.TEL_Limit_back_NC;
      A     L 20.0;
      A     "E      88.6";
      =     "INOUT".I_LIF.E88_6;
      A     L 20.0;
      A     "E      88.7";
      =     "INOUT".I_LIF.E88_7;
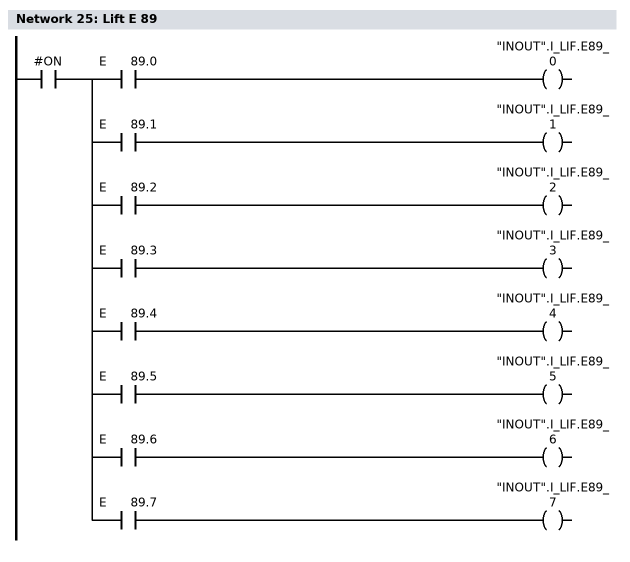
NETWORK
TITLE = Lift E 89
      A     #ON;
      =     L 20.0;
      A     L 20.0;
      A     "E      89.0";
      =     "INOUT".I_LIF.E89_0;
      A     L 20.0;
      A     "E      89.1";
      =     "INOUT".I_LIF.E89_1;
      A     L 20.0;
      A     "E      89.2";
      =     "INOUT".I_LIF.E89_2;
      A     L 20.0;
      A     "E      89.3";
      =     "INOUT".I_LIF.E89_3;
      A     L 20.0;
      A     "E      89.4";
      =     "INOUT".I_LIF.E89_4;
      A     L 20.0;
      A     "E      89.5";
      =     "INOUT".I_LIF.E89_5;
      A     L 20.0;
      A     "E      89.6";
      =     "INOUT".I_LIF.E89_6;
      A     L 20.0;
      A     "E      89.7";
      =     "INOUT".I_LIF.E89_7;
END_FUNCTION

FUNCTION "Outputs" : VOID	// FC 31
TITLE = Outputs
VERSION : 0.1
VAR_TEMP
  tmp_Retval : INT ;
  ON : BOOL ;
  OFF : BOOL ;
END_VAR
BEGIN
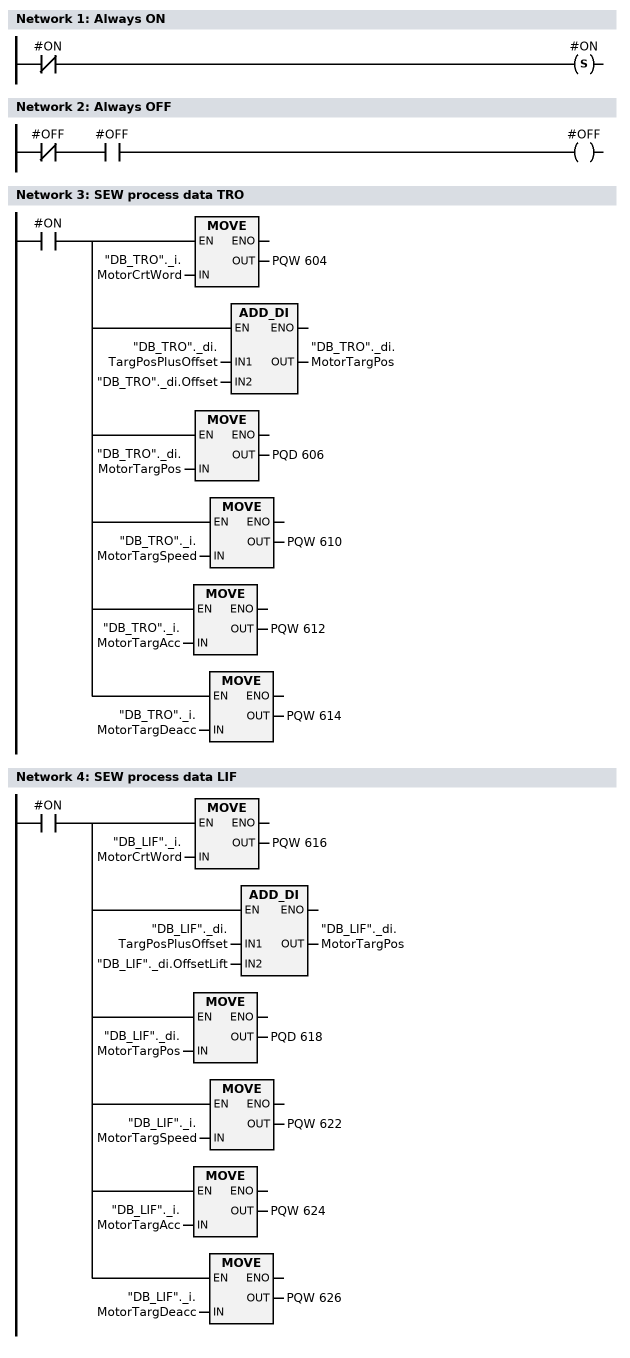
NETWORK
TITLE = Always ON
      AN    #ON;
      S     #ON;
NETWORK
TITLE = Always OFF
      AN    #OFF;
      A     #OFF;
      =     #OFF;
NETWORK
TITLE = SEW process data TRO
      A     #ON;
      =     L 3.0;
      A     L 3.0;
      JNB   _001;
      L     "DB_TRO"._i.MotorCrtWord;
      T     PQW 604;
_001: NOP   0;
      A     L 3.0;
      JNB   _002;
      L     "DB_TRO"._di.TargPosPlusOffset;
      L     "DB_TRO"._di.Offset;
      +D;
      T     "DB_TRO"._di.MotorTargPos;
_002: NOP   0;
      A     L 3.0;
      JNB   _003;
      L     "DB_TRO"._di.MotorTargPos;
      T     PQD 606;
_003: NOP   0;
      A     L 3.0;
      JNB   _004;
      L     "DB_TRO"._i.MotorTargSpeed;
      T     PQW 610;
_004: NOP   0;
      A     L 3.0;
      JNB   _005;
      L     "DB_TRO"._i.MotorTargAcc;
      T     PQW 612;
_005: NOP   0;
      A     L 3.0;
      JNB   _006;
      L     "DB_TRO"._i.MotorTargDeacc;
      T     PQW 614;
_006: NOP   0;
NETWORK
TITLE = SEW process data LIF
      A     #ON;
      =     L 3.0;
      A     L 3.0;
      JNB   _007;
      L     "DB_LIF"._i.MotorCrtWord;
      T     PQW 616;
_007: NOP   0;
      A     L 3.0;
      JNB   _008;
      L     "DB_LIF"._di.TargPosPlusOffset;
      L     "DB_LIF"._di.OffsetLift;
      +D;
      T     "DB_LIF"._di.MotorTargPos;
_008: NOP   0;
      A     L 3.0;
      JNB   _009;
      L     "DB_LIF"._di.MotorTargPos;
      T     PQD 618;
_009: NOP   0;
      A     L 3.0;
      JNB   _00a;
      L     "DB_LIF"._i.MotorTargSpeed;
      T     PQW 622;
_00a: NOP   0;
      A     L 3.0;
      JNB   _00b;
      L     "DB_LIF"._i.MotorTargAcc;
      T     PQW 624;
_00b: NOP   0;
      A     L 3.0;
      JNB   _00c;
      L     "DB_LIF"._i.MotorTargDeacc;
      T     PQW 626;
_00c: NOP   0;
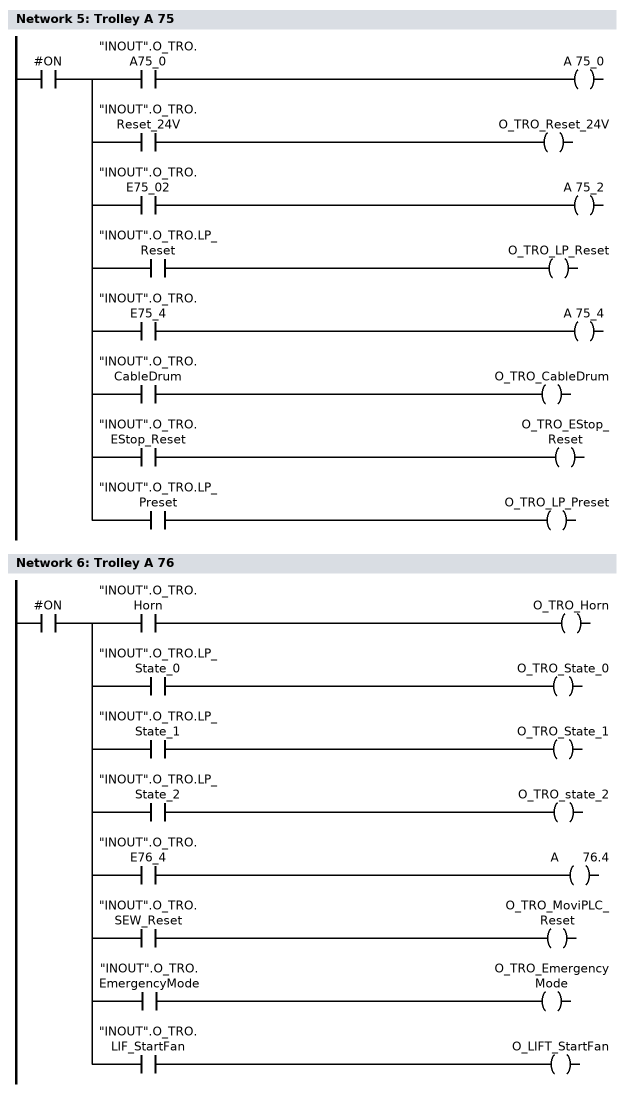
NETWORK
TITLE = Trolley A 75
      A     #ON;
      =     L 3.0;
      A     L 3.0;
      A     "INOUT".O_TRO.A75_0;
      =     "A 75_0";
      A     L 3.0;
      A     "INOUT".O_TRO.Reset_24V;
      =     "O_TRO_Reset_24V";
      A     L 3.0;
      A     "INOUT".O_TRO.E75_02;
      =     "A 75_2";
      A     L 3.0;
      A     "INOUT".O_TRO.LP_Reset;
      =     "O_TRO_LP_Reset";
      A     L 3.0;
      A     "INOUT".O_TRO.E75_4;
      =     "A 75_4";
      A     L 3.0;
      A     "INOUT".O_TRO.CableDrum;
      =     "O_TRO_CableDrum";
      A     L 3.0;
      A     "INOUT".O_TRO.EStop_Reset;
      =     "O_TRO_EStop_Reset";
      A     L 3.0;
      A     "INOUT".O_TRO.LP_Preset;
      =     "O_TRO_LP_Preset";
NETWORK
TITLE = Trolley A 76
      A     #ON;
      =     L 3.0;
      A     L 3.0;
      A     "INOUT".O_TRO.Horn;
      =     "O_TRO_Horn";
      A     L 3.0;
      A     "INOUT".O_TRO.LP_State_0;
      =     "O_TRO_State_0";
      A     L 3.0;
      A     "INOUT".O_TRO.LP_State_1;
      =     "O_TRO_State_1";
      A     L 3.0;
      A     "INOUT".O_TRO.LP_State_2;
      =     "O_TRO_state_2";
      A     L 3.0;
      A     "INOUT".O_TRO.E76_4;
      =     "A      76.4";
      A     L 3.0;
      A     "INOUT".O_TRO.SEW_Reset;
      =     "O_TRO_MoviPLC_Reset";
      A     L 3.0;
      A     "INOUT".O_TRO.EmergencyMode;
      =     "O_TRO_EmergencyMode";
      A     L 3.0;
      A     "INOUT".O_TRO.LIF_StartFan;
      =     "O_LIFT_StartFan";
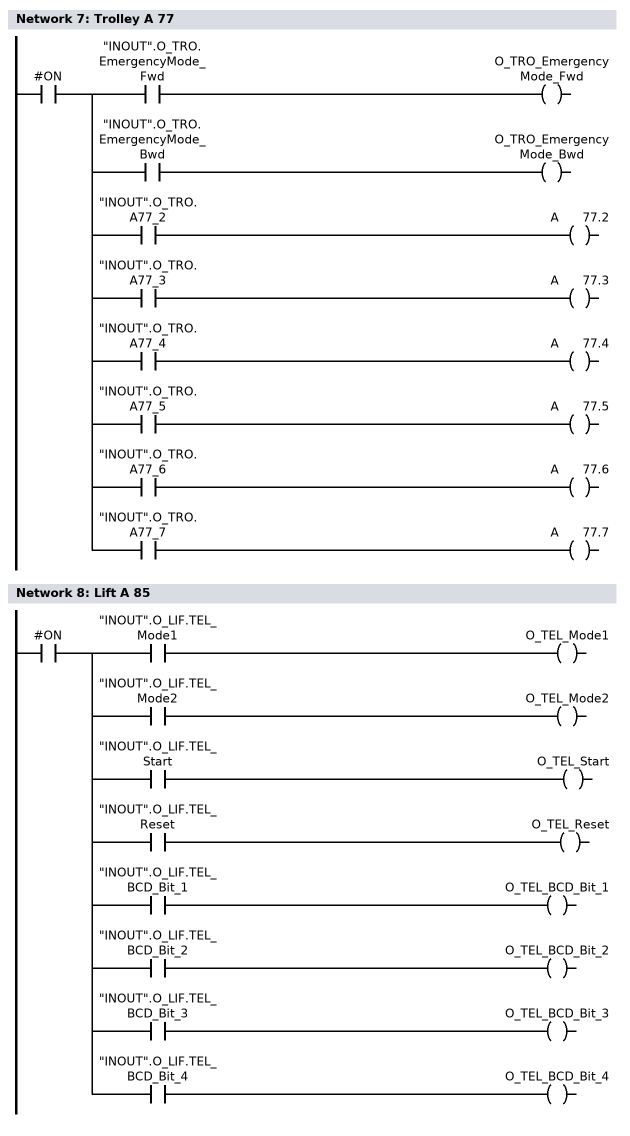
NETWORK
TITLE = Trolley A 77
      A     #ON;
      =     L 3.0;
      A     L 3.0;
      A     "INOUT".O_TRO.EmergencyMode_Fwd;
      =     "O_TRO_EmergencyMode_Fwd";
      A     L 3.0;
      A     "INOUT".O_TRO.EmergencyMode_Bwd;
      =     "O_TRO_EmergencyMode_Bwd";
      A     L 3.0;
      A     "INOUT".O_TRO.A77_2;
      =     "A      77.2";
      A     L 3.0;
      A     "INOUT".O_TRO.A77_3;
      =     "A      77.3";
      A     L 3.0;
      A     "INOUT".O_TRO.A77_4;
      =     "A      77.4";
      A     L 3.0;
      A     "INOUT".O_TRO.A77_5;
      =     "A      77.5";
      A     L 3.0;
      A     "INOUT".O_TRO.A77_6;
      =     "A      77.6";
      A     L 3.0;
      A     "INOUT".O_TRO.A77_7;
      =     "A      77.7";
NETWORK
TITLE = Lift A 85
      A     #ON;
      =     L 3.0;
      A     L 3.0;
      A     "INOUT".O_LIF.TEL_Mode1;
      =     "O_TEL_Mode1";
      A     L 3.0;
      A     "INOUT".O_LIF.TEL_Mode2;
      =     "O_TEL_Mode2";
      A     L 3.0;
      A     "INOUT".O_LIF.TEL_Start;
      =     "O_TEL_Start";
      A     L 3.0;
      A     "INOUT".O_LIF.TEL_Reset;
      =     "O_TEL_Reset";
      A     L 3.0;
      A     "INOUT".O_LIF.TEL_BCD_Bit_1;
      =     "O_TEL_BCD_Bit_1";
      A     L 3.0;
      A     "INOUT".O_LIF.TEL_BCD_Bit_2;
      =     "O_TEL_BCD_Bit_2";
      A     L 3.0;
      A     "INOUT".O_LIF.TEL_BCD_Bit_3;
      =     "O_TEL_BCD_Bit_3";
      A     L 3.0;
      A     "INOUT".O_LIF.TEL_BCD_Bit_4;
      =     "O_TEL_BCD_Bit_4";
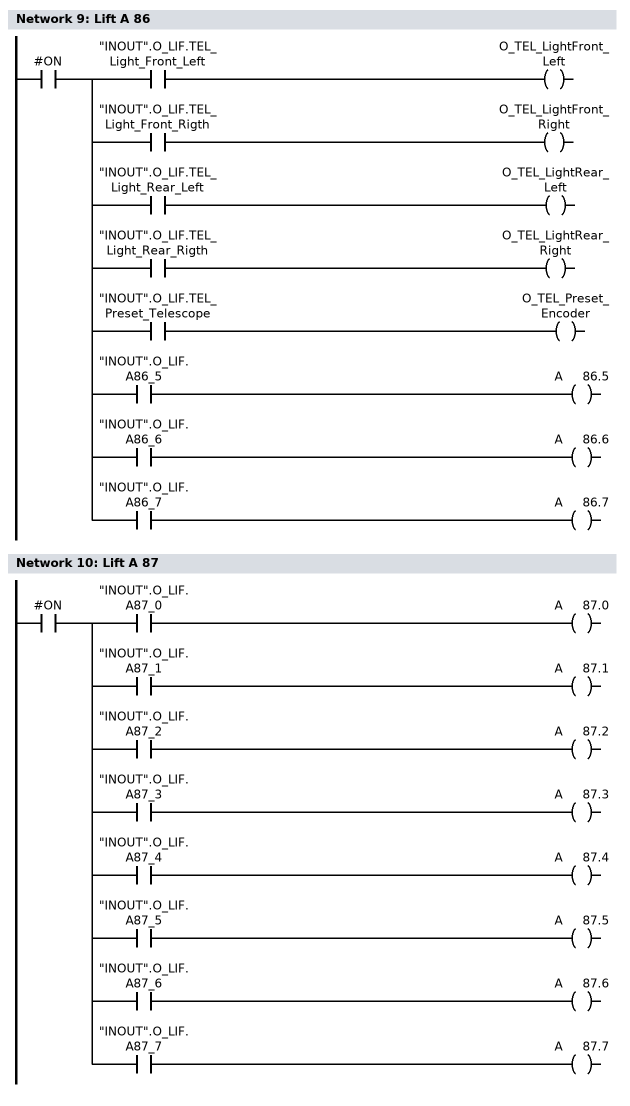
NETWORK
TITLE = Lift A 86
      A     #ON;
      =     L 3.0;
      A     L 3.0;
      A     "INOUT".O_LIF.TEL_Light_Front_Left;
      =     "O_TEL_LightFront_Left";
      A     L 3.0;
      A     "INOUT".O_LIF.TEL_Light_Front_Rigth;
      =     "O_TEL_LightFront_Right";
      A     L 3.0;
      A     "INOUT".O_LIF.TEL_Light_Rear_Left;
      =     "O_TEL_LightRear_Left";
      A     L 3.0;
      A     "INOUT".O_LIF.TEL_Light_Rear_Rigth;
      =     "O_TEL_LightRear_Right";
      A     L 3.0;
      A     "INOUT".O_LIF.TEL_Preset_Telescope;
      =     "O_TEL_Preset_Encoder";
      A     L 3.0;
      A     "INOUT".O_LIF.A86_5;
      =     "A     86.5";
      A     L 3.0;
      A     "INOUT".O_LIF.A86_6;
      =     "A     86.6";
      A     L 3.0;
      A     "INOUT".O_LIF.A86_7;
      =     "A     86.7";
NETWORK
TITLE = Lift A 87
      A     #ON;
      =     L 3.0;
      A     L 3.0;
      A     "INOUT".O_LIF.A87_0;
      =     "A     87.0";
      A     L 3.0;
      A     "INOUT".O_LIF.A87_1;
      =     "A     87.1";
      A     L 3.0;
      A     "INOUT".O_LIF.A87_2;
      =     "A     87.2";
      A     L 3.0;
      A     "INOUT".O_LIF.A87_3;
      =     "A     87.3";
      A     L 3.0;
      A     "INOUT".O_LIF.A87_4;
      =     "A     87.4";
      A     L 3.0;
      A     "INOUT".O_LIF.A87_5;
      =     "A     87.5";
      A     L 3.0;
      A     "INOUT".O_LIF.A87_6;
      =     "A     87.6";
      A     L 3.0;
      A     "INOUT".O_LIF.A87_7;
      =     "A     87.7";
END_FUNCTION

FUNCTION "MeasureSystem" : VOID	// FC 33
TITLE = Measure System
VERSION : 0.1
VAR_TEMP
  tmp_CircumOrder : DINT ;
  tmp_Circum : DINT ;
  tmp_Diff : DINT ;
  tmp_Measure : BOOL ;
  ON : BOOL ;
  OFF : BOOL ;
END_VAR
BEGIN
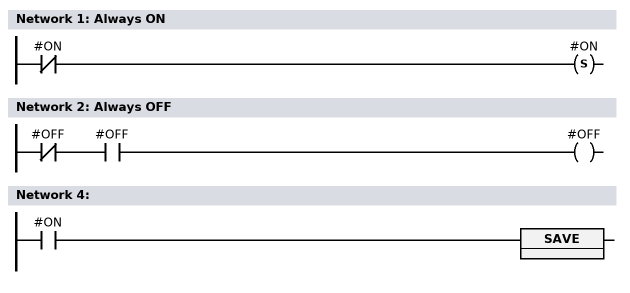
NETWORK
TITLE = Always ON
      AN    #ON;
      S     #ON;
NETWORK
TITLE = Always OFF
      AN    #OFF;
      A     #OFF;
      =     #OFF;
NETWORK
TITLE =
NETWORK
TITLE =
      A     #ON;
      SAVE;
END_FUNCTION

// FC 36: know-how protected block, not included

FUNCTION "Errors" : VOID	// FC 40
TITLE = Errors
VERSION : 0.1
VAR_TEMP
  ON : BOOL ;
  OFF : BOOL ;
END_VAR
BEGIN
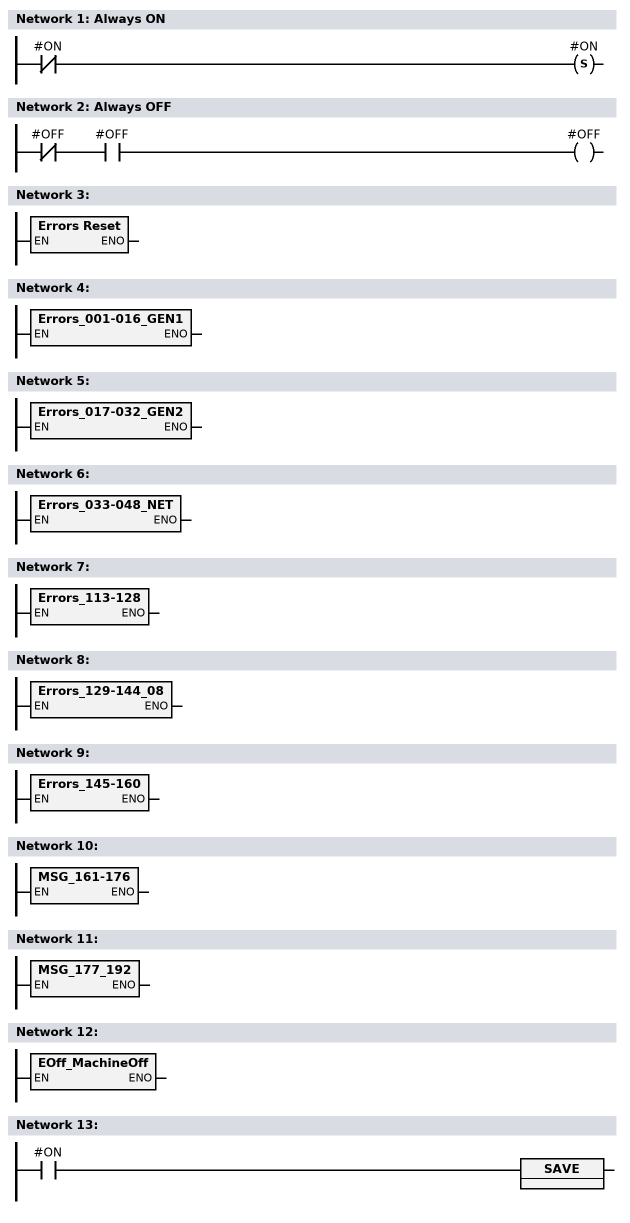
NETWORK
TITLE = Always ON
      AN    #ON;
      S     #ON;
NETWORK
TITLE = Always OFF
      AN    #OFF;
      A     #OFF;
      =     #OFF;
NETWORK
TITLE =
      CALL  "Errors Reset";
      NOP   0;
NETWORK
TITLE =
      CALL  "Errors_001-016_GEN1";
      NOP   0;
NETWORK
TITLE =
      CALL  "Errors_017-032_GEN2";
      NOP   0;
NETWORK
TITLE =
      CALL  "Errors_033-048_NET";
      NOP   0;
NETWORK
TITLE =
      CALL  "Errors_113-128";
      NOP   0;
NETWORK
TITLE =
      CALL  "Errors_129-144_08";
      NOP   0;
NETWORK
TITLE =
      CALL  "Errors_145-160";
      NOP   0;
NETWORK
TITLE =
      CALL  "MSG_161-176";
      NOP   0;
NETWORK
TITLE =
      CALL  "MSG_177_192";
      NOP   0;
NETWORK
TITLE =
      CALL  "EOff_MachineOff";
      NOP   0;
NETWORK
TITLE =
      A     #ON;
      SAVE;
END_FUNCTION

FUNCTION "Errors Reset" : VOID	// FC 41
TITLE = Errors Reset
VERSION : 0.1
VAR_TEMP
  tmp_RetVal : INT ;
  ON : BOOL ;
  OFF : BOOL ;
END_VAR
BEGIN
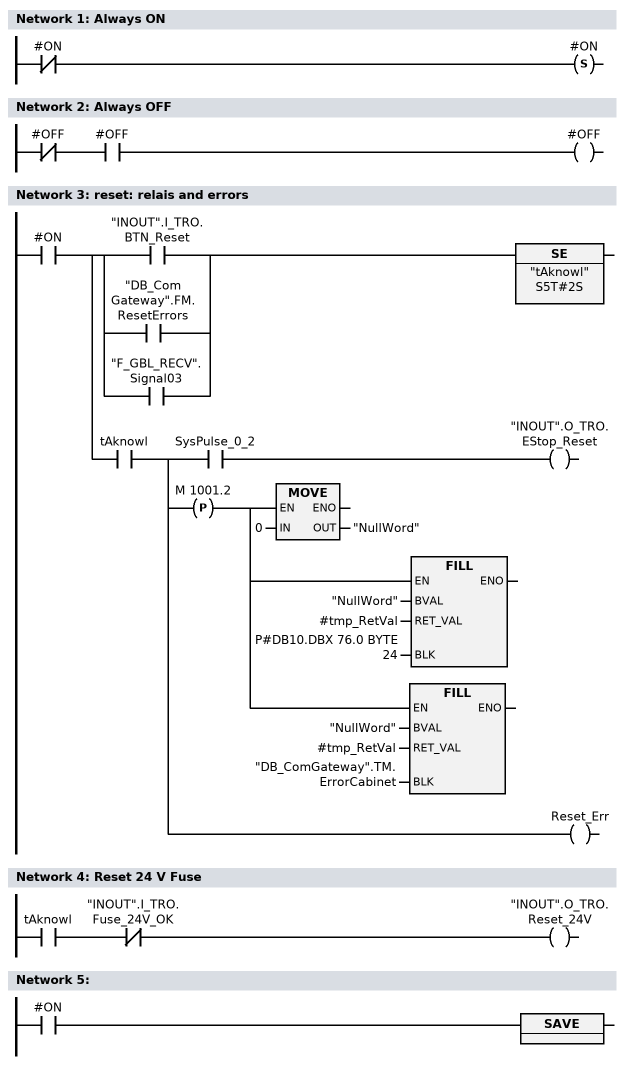
NETWORK
TITLE = Always ON
      AN    #ON;
      S     #ON;
NETWORK
TITLE = Always OFF
      AN    #OFF;
      A     #OFF;
      =     #OFF;
NETWORK
TITLE = reset: relais and errors
      A     #ON;
      =     L 3.0;
      A     L 3.0;
      A(;
      O     "INOUT".I_TRO.BTN_Reset;
      O     "DB_ComGateway".FM.ResetErrors;
      O     "F_GBL_RECV".Signal03;
      );
      L     S5T#2S;
      SE    "tAknowl";
      A     L 3.0;
      A     "tAknowl";
      =     L 3.1;
      A     L 3.1;
      A     "SysPulse_0_2";
      =     "INOUT".O_TRO.EStop_Reset;
      A     L 3.1;
      FP    M 1001.2;
      =     L 3.2;
      A     L 3.2;
      JNB   _001;
      L     0;
      T     "NullWord";
_001: NOP   0;
      A     L 3.2;
      JNB   _002;
      CALL  "FILL" (
           BVAL                     := "NullWord",
           RET_VAL                  := #tmp_RetVal,
           BLK                      := P#DB10.DBX 76.0 BYTE 24);
_002: NOP   0;
      A     L 3.2;
      JNB   _003;
      CALL  "FILL" (
           BVAL                     := "NullWord",
           RET_VAL                  := #tmp_RetVal,
           BLK                      := "DB_ComGateway".TM.ErrorCabinet);
_003: NOP   0;
      A     L 3.1;
      BLD   102;
      =     "Reset_Err";
NETWORK
TITLE = Reset 24 V Fuse
      A     "tAknowl";
      AN    "INOUT".I_TRO.Fuse_24V_OK;
      =     "INOUT".O_TRO.Reset_24V;
NETWORK
TITLE =
      A     #ON;
      SAVE;
END_FUNCTION

FUNCTION "Errors_001-016_GEN1" : VOID	// FC 42
TITLE = Errors GEN1
VERSION : 0.1
VAR_TEMP
  ON : BOOL ;
  OFF : BOOL ;
END_VAR
BEGIN
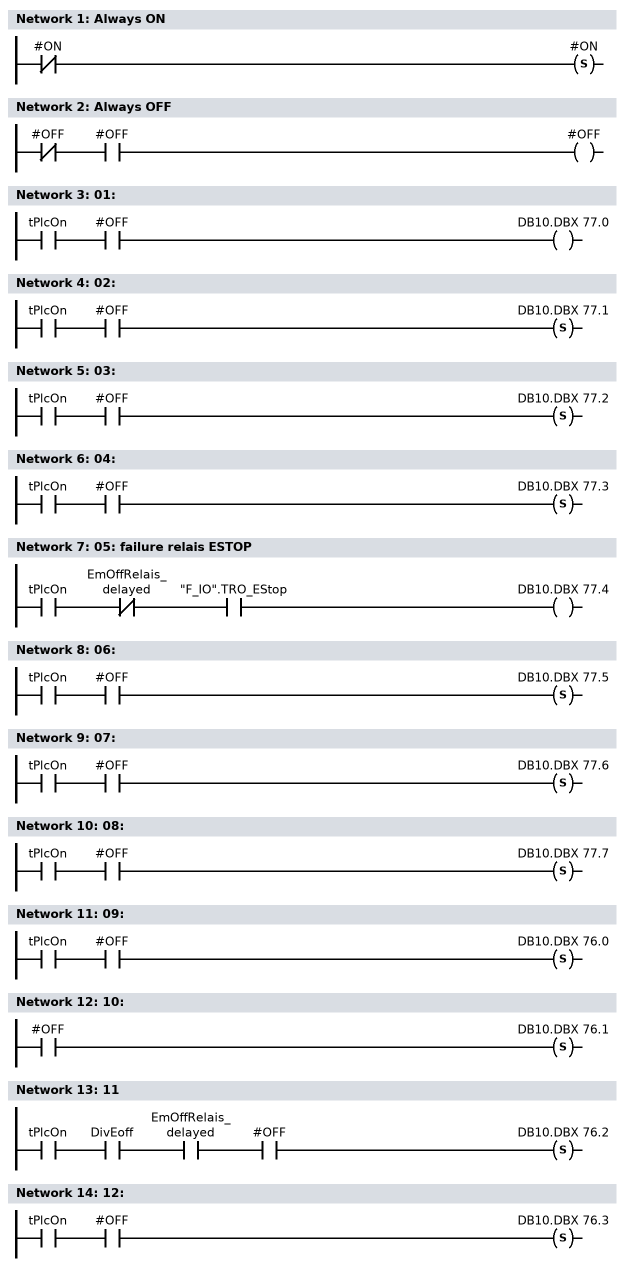
NETWORK
TITLE = Always ON
      AN    #ON;
      S     #ON;
NETWORK
TITLE = Always OFF
      AN    #OFF;
      A     #OFF;
      =     #OFF;
NETWORK
TITLE = 01:
      A     "tPlcOn";
      A     #OFF;
      =     DB10.DBX 77.0;
NETWORK
TITLE = 02:
      A     "tPlcOn";
      A     #OFF;
      S     DB10.DBX 77.1;
NETWORK
TITLE = 03:
      A     "tPlcOn";
      A     #OFF;
      S     DB10.DBX 77.2;
NETWORK
TITLE = 04:
      A     "tPlcOn";
      A     #OFF;
      S     DB10.DBX 77.3;
NETWORK
TITLE = 05: failure relais ESTOP
      A     "tPlcOn";
      AN    "EmOffRelais_delayed";
      A     "F_IO".TRO_EStop;
      =     DB10.DBX 77.4;
NETWORK
TITLE = 06:
      A     "tPlcOn";
      A     #OFF;
      S     DB10.DBX 77.5;
NETWORK
TITLE = 07:
      A     "tPlcOn";
      A     #OFF;
      S     DB10.DBX 77.6;
NETWORK
TITLE = 08:
      A     "tPlcOn";
      A     #OFF;
      S     DB10.DBX 77.7;
NETWORK
TITLE = 09:
      A     "tPlcOn";
      A     #OFF;
      S     DB10.DBX 76.0;
NETWORK
TITLE = 10:
      A     #OFF;
      S     DB10.DBX 76.1;
NETWORK
TITLE = 11
//10 eoff relais defekt
      A     "tPlcOn";
      A     "DivEoff";
      A     "EmOffRelais_delayed";
      A     #OFF;
      S     DB10.DBX 76.2;
NETWORK
TITLE = 12:
      A     "tPlcOn";
      A     #OFF;
      S     DB10.DBX 76.3;
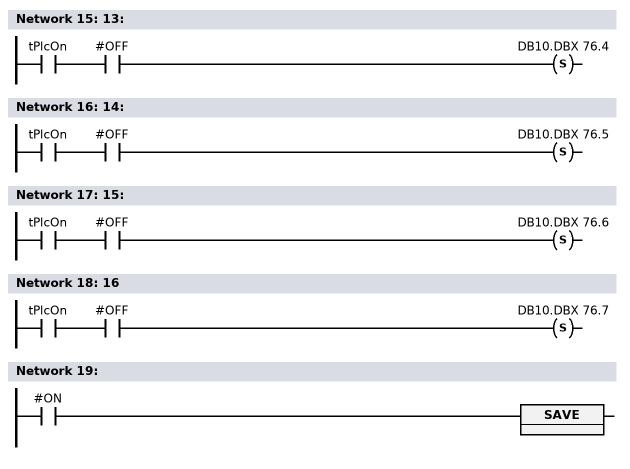
NETWORK
TITLE = 13:
      A     "tPlcOn";
      A     #OFF;
      S     DB10.DBX 76.4;
NETWORK
TITLE = 14:
      A     "tPlcOn";
      A     #OFF;
      S     DB10.DBX 76.5;
NETWORK
TITLE = 15:
      A     "tPlcOn";
      A     #OFF;
      S     DB10.DBX 76.6;
NETWORK
TITLE = 16
      A     "tPlcOn";
      A     #OFF;
      S     DB10.DBX 76.7;
NETWORK
TITLE =
      A     #ON;
      SAVE;
END_FUNCTION

FUNCTION "Errors_017-032_GEN2" : VOID	// FC 43
TITLE = Errors GEN2
VERSION : 0.1
VAR_TEMP
  ON : BOOL ;
  OFF : BOOL ;
END_VAR
BEGIN
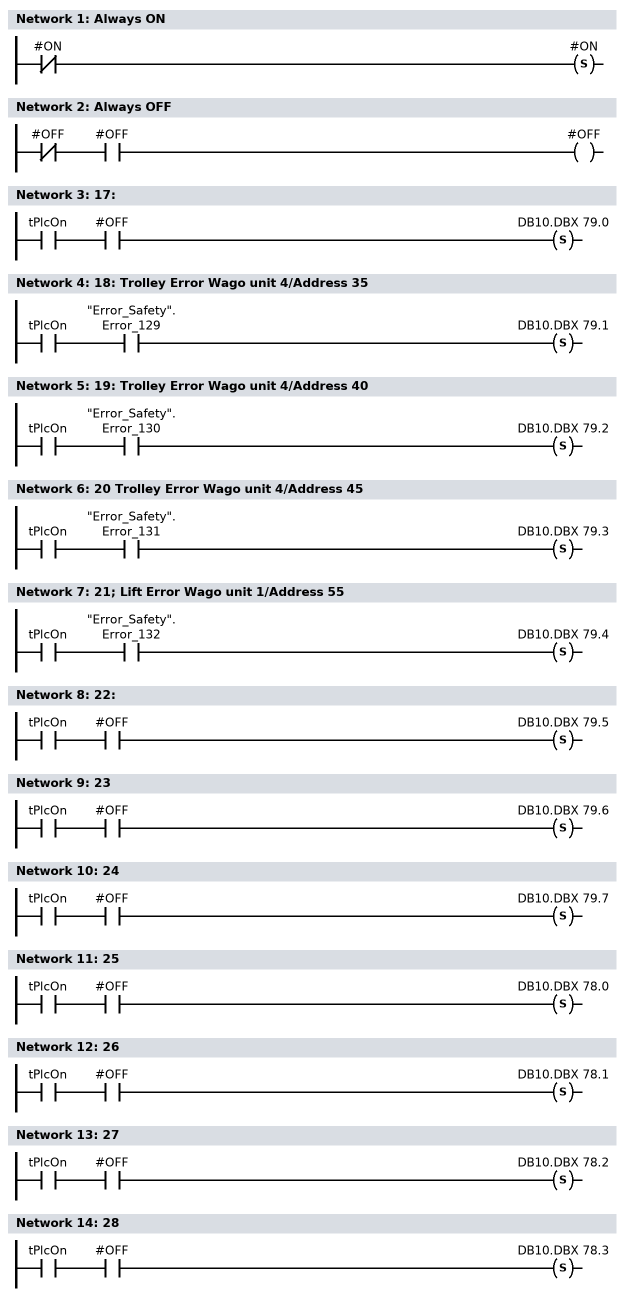
NETWORK
TITLE = Always ON
      AN    #ON;
      S     #ON;
NETWORK
TITLE = Always OFF
      AN    #OFF;
      A     #OFF;
      =     #OFF;
NETWORK
TITLE = 17:
      A     "tPlcOn";
      A     #OFF;
      S     DB10.DBX 79.0;
NETWORK
TITLE = 18: Trolley Error Wago unit 4/Address 35
      A     "tPlcOn";
      A     "Error_Safety".Error_129;
      S     DB10.DBX 79.1;
NETWORK
TITLE = 19: Trolley Error Wago unit 4/Address 40
      A     "tPlcOn";
      A     "Error_Safety".Error_130;
      S     DB10.DBX 79.2;
NETWORK
TITLE = 20 Trolley Error Wago unit 4/Address 45
      A     "tPlcOn";
      A     "Error_Safety".Error_131;
      S     DB10.DBX 79.3;
NETWORK
TITLE = 21; Lift Error Wago unit 1/Address 55
      A     "tPlcOn";
      A     "Error_Safety".Error_132;
      S     DB10.DBX 79.4;
NETWORK
TITLE = 22:
      A     "tPlcOn";
      A     #OFF;
      S     DB10.DBX 79.5;
NETWORK
TITLE = 23
      A     "tPlcOn";
      A     #OFF;
      S     DB10.DBX 79.6;
NETWORK
TITLE = 24
      A     "tPlcOn";
      A     #OFF;
      S     DB10.DBX 79.7;
NETWORK
TITLE = 25
      A     "tPlcOn";
      A     #OFF;
      S     DB10.DBX 78.0;
NETWORK
TITLE = 26
      A     "tPlcOn";
      A     #OFF;
      S     DB10.DBX 78.1;
NETWORK
TITLE = 27
      A     "tPlcOn";
      A     #OFF;
      S     DB10.DBX 78.2;
NETWORK
TITLE = 28
      A     "tPlcOn";
      A     #OFF;
      S     DB10.DBX 78.3;
